LIN {X -0.043,Y -388.097,Z 1443.709,A 0.000,B 0.000,C 90.000,E1 163.614} C_DIS
LIN {X -0.106,Y -389.112,Z 1443.709,A 0.000,B 0.000,C 90.000,E1 163.614} C_DIS
LIN {X 0.170,Y -391.805,Z 1443.708,A 0.000,B 0.000,C 90.000,E1 163.504} C_DIS
LIN {X 0.071,Y -393.632,Z 1443.708,A 0.000,B 0.000,C 90.000,E1 163.449} C_DIS
LIN {X 0.005,Y -396.516,Z 1443.707,A 0.000,B 0.000,C 90.000,E1 163.323} C_DIS
LIN {X 0.115,Y -399.461,Z 1443.707,A 0.000,B 0.000,C 90.000,E1 163.142} C_DIS
LIN {X -0.176,Y -405.694,Z 1443.704,A 0.000,B 0.000,C 90.000,E1 162.779} C_DIS
LIN {X -0.149,Y -411.913,Z 1443.702,A 0.000,B 0.000,C 90.000,E1 162.308} C_DIS
LIN {X 0.069,Y -418.024,Z 1443.699,A 0.000,B 0.000,C 90.000,E1 161.764} C_DIS
LIN {X -0.143,Y -430.224,Z 1443.693,A 0.000,B 0.000,C 90.000,E1 160.732} C_DIS
LIN {X 0.007,Y -445.761,Z 1443.686,A 0.000,B 0.000,C 90.000,E1 159.390} C_DIS
LIN {X 0.043,Y -457.905,Z 1443.680,A 0.000,B 0.000,C 90.000,E1 158.358} C_DIS
LIN {X -0.134,Y -466.994,Z 1443.676,A 0.000,B 0.000,C 90.000,E1 157.614} C_DIS
LIN {X 0.217,Y -474.540,Z 1443.672,A 0.000,B 0.000,C 90.000,E1 156.922} C_DIS
LIN {X -0.067,Y -483.447,Z 1443.668,A 0.000,B 0.000,C 90.000,E1 156.177} C_DIS
LIN {X 0.031,Y -493.492,Z 1443.662,A 0.000,B 0.000,C 90.000,E1 155.229} C_DIS
LIN {X 0.119,Y -500.398,Z 1443.659,A 0.000,B 0.000,C 90.000,E1 154.537} C_DIS
LIN {X -0.168,Y -505.638,Z 1443.656,A 0.000,B 0.000,C 90.000,E1 154.024} C_DIS
LIN {X -0.036,Y -510.716,Z 1443.652,A 0.000,B 0.000,C 90.000,E1 153.435} C_DIS
LIN {X -0.076,Y -514.384,Z 1443.650,A 0.000,B 0.000,C 90.000,E1 152.999} C_DIS
LIN {X -0.071,Y -518.865,Z 1443.647,A 0.000,B 0.000,C 90.000,E1 152.410} C_DIS
LIN {X -0.031,Y -522.887,Z 1443.643,A 0.000,B 0.000,C 90.000,E1 151.820} C_DIS
LIN {X -0.114,Y -527.207,Z 1443.639,A 0.000,B 0.000,C 90.000,E1 151.101} C_DIS
LIN {X -0.010,Y -530.289,Z 1443.636,A 0.000,B 0.000,C 90.000,E1 150.511} C_DIS
LIN {X -0.030,Y -533.682,Z 1443.632,A 0.000,B 0.000,C 90.000,E1 149.793} C_DIS
LIN {X 0.121,Y -536.153,Z 1443.629,A 0.000,B 0.000,C 90.000,E1 149.203} C_DIS
LIN {X -0.174,Y -538.356,Z 1443.626,A 0.000,B 0.000,C 90.000,E1 148.663} C_DIS
LIN {X 0.009,Y -541.283,Z 1443.621,A 0.000,B 0.000,C 90.000,E1 147.788} C_DIS
LIN {X 0.224,Y -543.843,Z 1443.616,A 0.000,B 0.000,C 90.000,E1 146.914} C_DIS
LIN {X 0.045,Y -546.875,Z 1443.610,A 0.000,B 0.000,C 90.000,E1 145.801} C_DIS
LIN {X -0.138,Y -548.886,Z 1443.605,A 0.000,B 0.000,C 90.000,E1 144.975} C_DIS
LIN {X -0.039,Y -550.081,Z 1443.602,A 0.000,B 0.000,C 90.000,E1 144.402} C_DIS
LIN {X 0.133,Y -551.642,Z 1443.598,A 0.000,B 0.000,C 90.000,E1 143.543} C_DIS
LIN {X -0.012,Y -552.949,Z 1443.593,A 0.000,B 0.000,C 90.000,E1 142.718} C_DIS
LIN {X -0.183,Y -554.507,Z 1443.587,A 0.000,B 0.000,C 90.000,E1 141.618} C_DIS
LIN {X 0.027,Y -555.474,Z 1443.582,A 0.000,B 0.000,C 90.000,E1 140.759} C_DIS
LIN {X -0.106,Y -556.824,Z 1443.574,A 0.000,B 0.000,C 90.000,E1 139.380} C_DIS
LIN {X -0.132,Y -558.199,Z 1443.565,A 0.000,B 0.000,C 90.000,E1 137.715} C_DIS
LIN {X 0.168,Y -559.249,Z 1443.557,A 0.000,B 0.000,C 90.000,E1 136.296} C_DIS
LIN {X 0.023,Y -559.895,Z 1443.551,A 0.000,B 0.000,C 90.000,E1 135.202} C_DIS
LIN {X 0.216,Y -560.297,Z 1443.547,A 0.000,B 0.000,C 90.000,E1 134.352} C_DIS
LIN {X -0.236,Y -560.810,Z 1443.539,A 0.000,B 0.000,C 90.000,E1 133.014} C_DIS
LIN {X 0.023,Y -561.097,Z 1443.533,A 0.000,B 0.000,C 90.000,E1 131.881} C_DIS
LIN {X 0.076,Y -561.154,Z 1443.524,A 0.000,B 0.000,C 90.000,E1 130.216} C_DIS
LIN {X 0.112,Y -561.234,Z 1443.516,A 0.000,B 0.000,C 90.000,E1 128.830} C_DIS
LIN {X 0.155,Y -561.226,Z 1443.508,A 0.000,B 0.000,C 90.000,E1 127.443} C_DIS
LIN {X -0.142,Y -561.158,Z 1443.500,A 0.000,B 0.000,C 90.000,E1 126.091} C_DIS
LIN {X 0.113,Y -560.907,Z 1443.491,A 0.000,B 0.000,C 90.000,E1 124.405} C_DIS
LIN {X -0.047,Y -560.612,Z 1443.484,A 0.000,B 0.000,C 90.000,E1 123.038} C_DIS
LIN {X 0.013,Y -560.329,Z 1443.470,A 0.000,B 0.000,C 90.000,E1 120.541} C_DIS
LIN {X 0.051,Y -560.806,Z 1443.454,A 0.000,B 0.000,C 90.000,E1 117.769} C_DIS
LIN {X -0.092,Y -561.432,Z 1443.444,A 0.000,B 0.000,C 90.000,E1 115.848} C_DIS
LIN {X -0.264,Y -561.973,Z 1443.434,A 0.000,B 0.000,C 90.000,E1 114.207} C_DIS
LIN {X 0.286,Y -562.387,Z 1443.427,A 0.000,B 0.000,C 90.000,E1 112.770} C_DIS
LIN {X 0.020,Y -563.124,Z 1443.416,A 0.000,B 0.000,C 90.000,E1 110.865} C_DIS
LIN {X -0.155,Y -563.887,Z 1443.408,A 0.000,B 0.000,C 90.000,E1 109.504} C_DIS
LIN {X 0.195,Y -564.616,Z 1443.405,A 0.000,B 0.000,C 90.000,E1 108.779} C_DIS
LIN {X -0.178,Y -565.734,Z 1443.402,A 0.000,B 0.000,C 90.000,E1 108.362} C_DIS
LIN {X 0.147,Y -567.188,Z 1443.400,A 0.000,B 0.000,C 90.000,E1 108.055} C_DIS
LIN {X -0.135,Y -568.209,Z 1443.400,A 0.000,B 0.000,C 90.000,E1 107.946} C_DIS
LIN {X 0.222,Y -571.023,Z 1443.398,A 0.000,B 0.000,C 90.000,E1 107.638} C_DIS
LIN {X -0.047,Y -580.628,Z 1443.394,A 0.000,B 0.000,C 90.000,E1 106.913} C_DIS
LIN {X 0.055,Y -584.581,Z 1443.392,A 0.000,B 0.000,C 90.000,E1 106.551} C_DIS
LIN {X -0.083,Y -587.115,Z 1443.391,A 0.000,B 0.000,C 90.000,E1 106.315} C_DIS
LIN {X -0.078,Y -591.677,Z 1443.388,A 0.000,B 0.000,C 90.000,E1 105.788} C_DIS
LIN {X -0.155,Y -592.571,Z 1443.387,A 0.000,B 0.000,C 90.000,E1 105.662} C_DIS
LIN {X -0.267,Y -596.101,Z 1443.383,A 0.000,B 0.000,C 90.000,E1 105.009} C_DIS
LIN {X 0.237,Y -596.677,Z 1443.383,A 0.000,B 0.000,C 90.000,E1 104.828} C_DIS
LIN {X 0.228,Y -597.980,Z 1443.380,A 0.000,B 0.000,C 90.000,E1 104.300} C_DIS
LIN {X -0.055,Y -599.497,Z 1443.375,A 0.000,B 0.000,C 90.000,E1 103.536} C_DIS
LIN {X -0.039,Y -600.150,Z 1443.372,A 0.000,B 0.000,C 90.000,E1 103.008} C_DIS
LIN {X -0.297,Y -600.745,Z 1443.368,A 0.000,B 0.000,C 90.000,E1 102.243} C_DIS
LIN {X 0.035,Y -600.724,Z 1443.364,A 0.000,B 0.000,C 90.000,E1 101.422} C_DIS
LIN {X -0.247,Y -600.676,Z 1443.362,A 0.000,B 0.000,C 90.000,E1 101.186} C_DIS
LIN {X -0.225,Y -599.926,Z 1443.359,A 0.000,B 0.000,C 90.000,E1 100.658} C_DIS
LIN {X -0.315,Y -598.816,Z 1443.356,A 0.000,B 0.000,C 90.000,E1 100.141} C_DIS
LIN {X -0.013,Y -598.181,Z 1443.355,A 0.000,B 0.000,C 90.000,E1 99.849} C_DIS
LIN {X -0.011,Y -596.569,Z 1443.352,A 0.000,B 0.000,C 90.000,E1 99.321} C_DIS
LIN {X -0.223,Y -593.855,Z 1443.348,A 0.000,B 0.000,C 90.000,E1 98.681} C_DIS
LIN {X 0.239,Y -591.207,Z 1443.345,A 0.000,B 0.000,C 90.000,E1 98.106} C_DIS
LIN {X 0.100,Y -588.095,Z 1443.342,A 0.000,B 0.000,C 90.000,E1 97.587} C_DIS
LIN {X -0.191,Y -583.595,Z 1443.339,A 0.000,B 0.000,C 90.000,E1 96.947} C_DIS
LIN {X 0.198,Y -579.504,Z 1443.336,A 0.000,B 0.000,C 90.000,E1 96.372} C_DIS
LIN {X -0.018,Y -574.862,Z 1443.333,A 0.000,B 0.000,C 90.000,E1 95.853} C_DIS
LIN {X -0.099,Y -572.597,Z 1443.330,A 0.000,B 0.000,C 90.000,E1 95.454} C_DIS
LIN {X 0.195,Y -571.361,Z 1443.329,A 0.000,B 0.000,C 90.000,E1 95.220} C_DIS
LIN {X 0.085,Y -571.073,Z 1443.329,A 0.000,B 0.000,C 90.000,E1 95.163} C_DIS
LIN {X 0.211,Y -570.540,Z 1443.327,A 0.000,B 0.000,C 90.000,E1 94.878} C_DIS
LIN {X -0.137,Y -570.023,Z 1443.324,A 0.000,B 0.000,C 90.000,E1 94.302} C_DIS
LIN {X 0.276,Y -570.225,Z 1443.319,A 0.000,B 0.000,C 90.000,E1 93.440} C_DIS
LIN {X -0.056,Y -571.455,Z 1443.310,A 0.000,B 0.000,C 90.000,E1 91.835} C_DIS
LIN {X -0.225,Y -573.087,Z 1443.300,A 0.000,B 0.000,C 90.000,E1 89.943} C_DIS
LIN {X -0.209,Y -575.053,Z 1443.287,A 0.000,B 0.000,C 90.000,E1 87.764} C_DIS
LIN {X -0.114,Y -577.038,Z 1443.276,A 0.000,B 0.000,C 90.000,E1 85.584} C_DIS
LIN {X 0.129,Y -579.039,Z 1443.263,A 0.000,B 0.000,C 90.000,E1 83.394} C_DIS
LIN {X -0.084,Y -580.371,Z 1443.256,A 0.000,B 0.000,C 90.000,E1 82.064} C_DIS
LIN {X -0.280,Y -581.712,Z 1443.248,A 0.000,B 0.000,C 90.000,E1 80.735} C_DIS
LIN {X -0.228,Y -583.857,Z 1443.236,A 0.000,B 0.000,C 90.000,E1 78.578} C_DIS
LIN {X 0.166,Y -584.968,Z 1443.230,A 0.000,B 0.000,C 90.000,E1 77.465} C_DIS
LIN {X 0.165,Y -586.431,Z 1443.220,A 0.000,B 0.000,C 90.000,E1 75.589} C_DIS
LIN {X 0.159,Y -587.187,Z 1443.214,A 0.000,B 0.000,C 90.000,E1 74.519} C_DIS
LIN {X 0.251,Y -588.124,Z 1443.205,A 0.000,B 0.000,C 90.000,E1 72.906} C_DIS
LIN {X -0.116,Y -588.784,Z 1443.199,A 0.000,B 0.000,C 90.000,E1 71.873} C_DIS
LIN {X -0.133,Y -589.718,Z 1443.189,A 0.000,B 0.000,C 90.000,E1 70.007} C_DIS
LIN {X 0.155,Y -590.890,Z 1443.177,A 0.000,B 0.000,C 90.000,E1 67.847} C_DIS
LIN {X -0.064,Y -591.621,Z 1443.170,A 0.000,B 0.000,C 90.000,E1 66.538} C_DIS
LIN {X -0.321,Y -593.633,Z 1443.153,A 0.000,B 0.000,C 90.000,E1 63.640} C_DIS
LIN {X -0.075,Y -594.193,Z 1443.149,A 0.000,B 0.000,C 90.000,E1 62.820} C_DIS
LIN {X -0.243,Y -595.838,Z 1443.137,A 0.000,B 0.000,C 90.000,E1 60.717} C_DIS
LIN {X -0.306,Y -596.762,Z 1443.131,A 0.000,B 0.000,C 90.000,E1 59.665} C_DIS
LIN {X -0.143,Y -597.955,Z 1443.124,A 0.000,B 0.000,C 90.000,E1 58.329} C_DIS
LIN {X 0.128,Y -598.911,Z 1443.118,A 0.000,B 0.000,C 90.000,E1 57.248} C_DIS
LIN {X 0.052,Y -600.312,Z 1443.109,A 0.000,B 0.000,C 90.000,E1 55.674} C_DIS
LIN {X -0.149,Y -601.697,Z 1443.101,A 0.000,B 0.000,C 90.000,E1 54.116} C_DIS
LIN {X -0.067,Y -602.999,Z 1443.090,A 0.000,B 0.000,C 90.000,E1 52.271} C_DIS
LIN {X -0.370,Y -603.736,Z 1443.085,A 0.000,B 0.000,C 90.000,E1 51.251} C_DIS
LIN {X 0.233,Y -604.562,Z 1443.076,A 0.000,B 0.000,C 90.000,E1 49.622} C_DIS
LIN {X -0.121,Y -604.812,Z 1443.070,A 0.000,B 0.000,C 90.000,E1 48.609} C_DIS
LIN {X -0.165,Y -605.143,Z 1443.060,A 0.000,B 0.000,C 90.000,E1 46.782} C_DIS
LIN {X -0.285,Y -605.195,Z 1443.053,A 0.000,B 0.000,C 90.000,E1 45.486} C_DIS
LIN {X 0.183,Y -605.142,Z 1443.050,A 0.000,B 0.000,C 90.000,E1 44.919} C_DIS
LIN {X -0.399,Y -604.870,Z 1443.045,A 0.000,B 0.000,C 90.000,E1 44.190} C_DIS
LIN {X 0.112,Y -604.301,Z 1443.040,A 0.000,B 0.000,C 90.000,E1 43.095} C_DIS
LIN {X 0.413,Y -603.357,Z 1443.032,A 0.000,B 0.000,C 90.000,E1 41.757} C_DIS
LIN {X 0.249,Y -602.682,Z 1443.028,A 0.000,B 0.000,C 90.000,E1 40.987} C_DIS
LIN {X -0.065,Y -601.561,Z 1443.022,A 0.000,B 0.000,C 90.000,E1 39.967} C_DIS
LIN {X -0.227,Y -599.921,Z 1443.015,A 0.000,B 0.000,C 90.000,E1 38.669} C_DIS
LIN {X -0.098,Y -598.436,Z 1443.009,A 0.000,B 0.000,C 90.000,E1 37.604} C_DIS
LIN {X 0.139,Y -597.159,Z 1443.005,A 0.000,B 0.000,C 90.000,E1 36.790} C_DIS
LIN {X 0.231,Y -595.164,Z 1442.999,A 0.000,B 0.000,C 90.000,E1 35.724} C_DIS
LIN {X 0.073,Y -593.383,Z 1442.994,A 0.000,B 0.000,C 90.000,E1 34.945} C_DIS
LIN {X -0.230,Y -590.841,Z 1442.988,A 0.000,B 0.000,C 90.000,E1 33.913} C_DIS
LIN {X -0.069,Y -587.912,Z 1442.982,A 0.000,B 0.000,C 90.000,E1 32.832} C_DIS
LIN {X 0.183,Y -585.485,Z 1442.978,A 0.000,B 0.000,C 90.000,E1 32.005} C_DIS
LIN {X 0.232,Y -583.740,Z 1442.975,A 0.000,B 0.000,C 90.000,E1 31.465} C_DIS
LIN {X 0.130,Y -580.685,Z 1442.970,A 0.000,B 0.000,C 90.000,E1 30.669} C_DIS
LIN {X 0.072,Y -577.807,Z 1442.967,A 0.000,B 0.000,C 90.000,E1 30.001} C_DIS
LIN {X -0.173,Y -573.342,Z 1442.962,A 0.000,B 0.000,C 90.000,E1 29.077} C_DIS
LIN {X 0.197,Y -569.830,Z 1442.958,A 0.000,B 0.000,C 90.000,E1 28.359} C_DIS
LIN {X -0.146,Y -566.821,Z 1442.955,A 0.000,B 0.000,C 90.000,E1 27.847} C_DIS
LIN {X -0.028,Y -561.226,Z 1442.949,A 0.000,B 0.000,C 90.000,E1 26.873} C_DIS
LIN {X -0.127,Y -556.006,Z 1442.945,A 0.000,B 0.000,C 90.000,E1 26.052} C_DIS
LIN {X 0.293,Y -553.280,Z 1442.942,A 0.000,B 0.000,C 90.000,E1 25.591} C_DIS
LIN {X -0.156,Y -549.389,Z 1442.939,A 0.000,B 0.000,C 90.000,E1 25.079} C_DIS
LIN {X 0.242,Y -544.155,Z 1442.935,A 0.000,B 0.000,C 90.000,E1 24.335} C_DIS
LIN {X -0.138,Y -540.821,Z 1442.933,A 0.000,B 0.000,C 90.000,E1 23.951} C_DIS
LIN {X 0.182,Y -534.920,Z 1442.929,A 0.000,B 0.000,C 90.000,E1 23.206} C_DIS
LIN {X -0.196,Y -527.495,Z 1442.924,A 0.000,B 0.000,C 90.000,E1 22.386} C_DIS
LIN {X 0.203,Y -518.579,Z 1442.919,A 0.000,B 0.000,C 90.000,E1 21.354} C_DIS
LIN {X 0.160,Y -509.329,Z 1442.913,A 0.000,B 0.000,C 90.000,E1 20.375} C_DIS
LIN {X -0.060,Y -498.393,Z 1442.907,A 0.000,B 0.000,C 90.000,E1 19.268} C_DIS
LIN {X 0.009,Y -478.216,Z 1442.895,A 0.000,B 0.000,C 90.000,E1 17.166} C_DIS
LIN {X 0.259,Y -464.739,Z 1442.887,A 0.000,B 0.000,C 90.000,E1 15.662} C_DIS
LIN {X 0.014,Y -460.341,Z 1442.885,A 0.000,B 0.000,C 90.000,E1 15.245} C_DIS
LIN {X -0.012,Y -455.773,Z 1442.882,A 0.000,B 0.000,C 90.000,E1 14.828} C_DIS
LIN {X 0.032,Y -450.844,Z 1442.880,A 0.000,B 0.000,C 90.000,E1 14.426} C_DIS
LIN {X 0.002,Y -447.084,Z 1442.879,A 0.000,B 0.000,C 90.000,E1 14.189} C_DIS
LIN {X 0.033,Y -444.395,Z 1442.878,A 0.000,B 0.000,C 90.000,E1 14.064} C_DIS
LIN {X 0.098,Y -442.520,Z 1442.878,A 0.000,B 0.000,C 90.000,E1 14.008} C_DIS
LIN {X 0.070,Y -442.170,Z 1442.878,A 0.000,B 0.000,C 90.000,E1 14.008} C_DIS
LIN {X 0.034,Y -369.502,Z 1442.878,A 0.000,B 0.000,C 90.000,E1 14.008} C_DIS
LIN {X 0.102,Y -366.485,Z 1442.855,A 0.000,B 0.000,C 90.000,E1 9.905} C_DIS
LIN {X 0.038,Y -361.787,Z 1442.822,A 0.000,B 0.000,C 90.000,E1 3.955} C_DIS
LIN {X -0.077,Y -360.901,Z 1442.801,A 0.000,B 0.000,C 90.000,E1 0.229} C_DIS
LIN {X -0.053,Y -359.426,Z 1442.770,A 0.000,B 0.000,C 90.000,E1 354.546} C_DIS
LIN {X 0.070,Y -358.890,Z 1442.759,A 0.000,B 0.000,C 90.000,E1 352.648} C_DIS
LIN {X -0.020,Y -359.563,Z 1442.726,A 0.000,B 0.000,C 90.000,E1 346.645} C_DIS
LIN {X 0.001,Y -361.801,Z 1442.684,A 0.000,B 0.000,C 90.000,E1 339.135} C_DIS
LIN {X -0.154,Y -362.053,Z 1442.680,A 0.000,B 0.000,C 90.000,E1 338.411} C_DIS
LIN {X 0.189,Y -365.980,Z 1442.643,A 0.000,B 0.000,C 90.000,E1 331.641} C_DIS
LIN {X 0.029,Y -366.387,Z 1442.639,A 0.000,B 0.000,C 90.000,E1 330.923} C_DIS
LIN {X -0.031,Y -371.355,Z 1442.604,A 0.000,B 0.000,C 90.000,E1 324.642} C_DIS
LIN {X -0.043,Y -371.766,Z 1442.602,A 0.000,B 0.000,C 90.000,E1 324.276} C_DIS
LIN {X 0.013,Y -377.358,Z 1442.567,A 0.000,B 0.000,C 90.000,E1 318.038} C_DIS
LIN {X 0.012,Y -378.235,Z 1442.563,A 0.000,B 0.000,C 90.000,E1 317.310} C_DIS
LIN {X 0.002,Y -383.940,Z 1442.531,A 0.000,B 0.000,C 90.000,E1 311.515} C_DIS
LIN {X 0.088,Y -384.893,Z 1442.527,A 0.000,B 0.000,C 90.000,E1 310.782} C_DIS
LIN {X 0.262,Y -390.610,Z 1442.495,A 0.000,B 0.000,C 90.000,E1 305.025} C_DIS
LIN {X 0.106,Y -391.104,Z 1442.493,A 0.000,B 0.000,C 90.000,E1 304.692} C_DIS
LIN {X 0.022,Y -391.648,Z 1442.489,A 0.000,B 0.000,C 90.000,E1 303.992} C_DIS
LIN {X -0.080,Y -396.825,Z 1442.459,A 0.000,B 0.000,C 90.000,E1 298.693} C_DIS
LIN {X -0.210,Y -397.120,Z 1442.457,A 0.000,B 0.000,C 90.000,E1 298.359} C_DIS
LIN {X -0.055,Y -401.597,Z 1442.426,A 0.000,B 0.000,C 90.000,E1 292.717} C_DIS
LIN {X 0.222,Y -404.659,Z 1442.395,A 0.000,B 0.000,C 90.000,E1 287.094} C_DIS
LIN {X -0.079,Y -404.735,Z 1442.391,A 0.000,B 0.000,C 90.000,E1 286.441} C_DIS
LIN {X 0.214,Y -406.099,Z 1442.364,A 0.000,B 0.000,C 90.000,E1 281.535} C_DIS
LIN {X -0.176,Y -406.094,Z 1442.362,A 0.000,B 0.000,C 90.000,E1 281.243} C_DIS
LIN {X -0.097,Y -405.680,Z 1442.333,A 0.000,B 0.000,C 90.000,E1 276.024} C_DIS
LIN {X -0.165,Y -405.058,Z 1442.328,A 0.000,B 0.000,C 90.000,E1 274.992} C_DIS
LIN {X -0.060,Y -403.497,Z 1442.304,A 0.000,B 0.000,C 90.000,E1 270.802} C_DIS
LIN {X -0.092,Y -403.288,Z 1442.302,A 0.000,B 0.000,C 90.000,E1 270.458} C_DIS
LIN {X 0.091,Y -398.931,Z 1442.271,A 0.000,B 0.000,C 90.000,E1 264.837} C_DIS
LIN {X -0.040,Y -393.108,Z 1442.242,A 0.000,B 0.000,C 90.000,E1 259.567} C_DIS
LIN {X -0.079,Y -392.835,Z 1442.240,A 0.000,B 0.000,C 90.000,E1 259.218} C_DIS
LIN {X 0.034,Y -385.993,Z 1442.212,A 0.000,B 0.000,C 90.000,E1 254.212} C_DIS
LIN {X -0.026,Y -385.267,Z 1442.208,A 0.000,B 0.000,C 90.000,E1 253.504} C_DIS
LIN {X -0.004,Y -384.768,Z 1442.206,A 0.000,B 0.000,C 90.000,E1 253.142} C_DIS
LIN {X 0.221,Y -377.973,Z 1442.182,A 0.000,B 0.000,C 90.000,E1 248.773} C_DIS
LIN {X -0.044,Y -376.233,Z 1442.174,A 0.000,B 0.000,C 90.000,E1 247.358} C_DIS
LIN {X 0.057,Y -374.944,Z 1442.170,A 0.000,B 0.000,C 90.000,E1 246.613} C_DIS
LIN {X -0.208,Y -368.417,Z 1442.148,A 0.000,B 0.000,C 90.000,E1 242.615} C_DIS
LIN {X 0.097,Y -366.047,Z 1442.137,A 0.000,B 0.000,C 90.000,E1 240.717} C_DIS
LIN {X 0.004,Y -359.196,Z 1442.115,A 0.000,B 0.000,C 90.000,E1 236.628} C_DIS
LIN {X 0.021,Y -355.842,Z 1442.100,A 0.000,B 0.000,C 90.000,E1 233.989} C_DIS
LIN {X -0.173,Y -348.793,Z 1442.075,A 0.000,B 0.000,C 90.000,E1 229.461} C_DIS
LIN {X -0.097,Y -346.185,Z 1442.062,A 0.000,B 0.000,C 90.000,E1 227.148} C_DIS
LIN {X -0.088,Y -345.065,Z 1442.058,A 0.000,B 0.000,C 90.000,E1 226.377} C_DIS
LIN {X 0.094,Y -338.586,Z 1442.030,A 0.000,B 0.000,C 90.000,E1 221.310} C_DIS
LIN {X 0.094,Y -336.840,Z 1442.019,A 0.000,B 0.000,C 90.000,E1 219.358} C_DIS
LIN {X 0.014,Y -330.861,Z 1441.988,A 0.000,B 0.000,C 90.000,E1 213.865} C_DIS
LIN {X 0.149,Y -329.296,Z 1441.975,A 0.000,B 0.000,C 90.000,E1 211.465} C_DIS
LIN {X -0.154,Y -324.669,Z 1441.942,A 0.000,B 0.000,C 90.000,E1 205.540} C_DIS
LIN {X 0.174,Y -323.837,Z 1441.928,A 0.000,B 0.000,C 90.000,E1 203.078} C_DIS
LIN {X -0.017,Y -321.124,Z 1441.881,A 0.000,B 0.000,C 90.000,E1 194.662} C_DIS
LIN {X 0.138,Y -320.932,Z 1441.877,A 0.000,B 0.000,C 90.000,E1 193.828} C_DIS
LIN {X -0.076,Y -321.562,Z 1441.832,A 0.000,B 0.000,C 90.000,E1 185.796} C_DIS
LIN {X -0.143,Y -324.415,Z 1441.790,A 0.000,B 0.000,C 90.000,E1 178.165} C_DIS
LIN {X -0.141,Y -325.376,Z 1441.783,A 0.000,B 0.000,C 90.000,E1 176.963} C_DIS
LIN {X -0.100,Y -329.112,Z 1441.750,A 0.000,B 0.000,C 90.000,E1 170.971} C_DIS
LIN {X 0.061,Y -334.260,Z 1441.726,A 0.000,B 0.000,C 90.000,E1 166.589} C_DIS
LIN {X 0.067,Y -335.488,Z 1441.719,A 0.000,B 0.000,C 90.000,E1 165.408} C_DIS
LIN {X -0.119,Y -336.681,Z 1441.713,A 0.000,B 0.000,C 90.000,E1 164.338} C_DIS
LIN {X -0.154,Y -381.447,Z 1441.713,A 0.000,B 0.000,C 90.000,E1 164.338} C_DIS
LIN {X 0.204,Y -384.725,Z 1441.713,A 0.000,B 0.000,C 90.000,E1 164.212} C_DIS
LIN {X -0.022,Y -386.911,Z 1441.712,A 0.000,B 0.000,C 90.000,E1 164.157} C_DIS
LIN {X -0.146,Y -389.736,Z 1441.711,A 0.000,B 0.000,C 90.000,E1 164.031} C_DIS
LIN {X 0.097,Y -395.861,Z 1441.709,A 0.000,B 0.000,C 90.000,E1 163.614} C_DIS
LIN {X -0.141,Y -402.081,Z 1441.707,A 0.000,B 0.000,C 90.000,E1 163.196} C_DIS
LIN {X 0.031,Y -408.356,Z 1441.704,A 0.000,B 0.000,C 90.000,E1 162.670} C_DIS
LIN {X 0.045,Y -422.169,Z 1441.697,A 0.000,B 0.000,C 90.000,E1 161.456} C_DIS
LIN {X -0.198,Y -434.491,Z 1441.691,A 0.000,B 0.000,C 90.000,E1 160.423} C_DIS
LIN {X 0.067,Y -448.418,Z 1441.685,A 0.000,B 0.000,C 90.000,E1 159.209} C_DIS
LIN {X 0.281,Y -460.594,Z 1441.679,A 0.000,B 0.000,C 90.000,E1 158.156} C_DIS
LIN {X -0.085,Y -471.156,Z 1441.674,A 0.000,B 0.000,C 90.000,E1 157.305} C_DIS
LIN {X 0.223,Y -483.026,Z 1441.668,A 0.000,B 0.000,C 90.000,E1 156.230} C_DIS
LIN {X -0.253,Y -491.639,Z 1441.664,A 0.000,B 0.000,C 90.000,E1 155.485} C_DIS
LIN {X -0.063,Y -497.243,Z 1441.661,A 0.000,B 0.000,C 90.000,E1 154.921} C_DIS
LIN {X 0.015,Y -502.740,Z 1441.658,A 0.000,B 0.000,C 90.000,E1 154.357} C_DIS
LIN {X -0.077,Y -506.692,Z 1441.655,A 0.000,B 0.000,C 90.000,E1 153.948} C_DIS
LIN {X -0.161,Y -511.719,Z 1441.652,A 0.000,B 0.000,C 90.000,E1 153.384} C_DIS
LIN {X -0.003,Y -515.332,Z 1441.650,A 0.000,B 0.000,C 90.000,E1 152.922} C_DIS
LIN {X -0.229,Y -519.733,Z 1441.646,A 0.000,B 0.000,C 90.000,E1 152.359} C_DIS
LIN {X -0.186,Y -523.691,Z 1441.643,A 0.000,B 0.000,C 90.000,E1 151.769} C_DIS
LIN {X -0.110,Y -527.162,Z 1441.640,A 0.000,B 0.000,C 90.000,E1 151.179} C_DIS
LIN {X -0.008,Y -530.281,Z 1441.637,A 0.000,B 0.000,C 90.000,E1 150.589} C_DIS
LIN {X -0.030,Y -533.716,Z 1441.633,A 0.000,B 0.000,C 90.000,E1 149.871} C_DIS
LIN {X 0.118,Y -536.208,Z 1441.630,A 0.000,B 0.000,C 90.000,E1 149.282} C_DIS
LIN {X -0.179,Y -538.438,Z 1441.626,A 0.000,B 0.000,C 90.000,E1 148.742} C_DIS
LIN {X 0.003,Y -541.355,Z 1441.622,A 0.000,B 0.000,C 90.000,E1 147.867} C_DIS
LIN {X -0.240,Y -543.932,Z 1441.617,A 0.000,B 0.000,C 90.000,E1 147.041} C_DIS
LIN {X 0.036,Y -546.954,Z 1441.610,A 0.000,B 0.000,C 90.000,E1 145.881} C_DIS
LIN {X -0.149,Y -548.980,Z 1441.606,A 0.000,B 0.000,C 90.000,E1 145.055} C_DIS
LIN {X 0.003,Y -550.716,Z 1441.601,A 0.000,B 0.000,C 90.000,E1 144.196} C_DIS
LIN {X 0.181,Y -552.207,Z 1441.596,A 0.000,B 0.000,C 90.000,E1 143.336} C_DIS
LIN {X -0.333,Y -553.829,Z 1441.590,A 0.000,B 0.000,C 90.000,E1 142.271} C_DIS
LIN {X 0.292,Y -555.266,Z 1441.584,A 0.000,B 0.000,C 90.000,E1 141.090} C_DIS
LIN {X -0.195,Y -556.619,Z 1441.576,A 0.000,B 0.000,C 90.000,E1 139.747} C_DIS
LIN {X -0.220,Y -558.014,Z 1441.567,A 0.000,B 0.000,C 90.000,E1 138.081} C_DIS
LIN {X 0.081,Y -559.071,Z 1441.559,A 0.000,B 0.000,C 90.000,E1 136.662} C_DIS
LIN {X -0.058,Y -559.788,Z 1441.553,A 0.000,B 0.000,C 90.000,E1 135.567} C_DIS
LIN {X 0.201,Y -560.311,Z 1441.547,A 0.000,B 0.000,C 90.000,E1 134.433} C_DIS
LIN {X 0.132,Y -560.797,Z 1441.539,A 0.000,B 0.000,C 90.000,E1 133.056} C_DIS
LIN {X -0.035,Y -561.010,Z 1441.535,A 0.000,B 0.000,C 90.000,E1 132.243} C_DIS
LIN {X -0.149,Y -561.120,Z 1441.529,A 0.000,B 0.000,C 90.000,E1 131.148} C_DIS
LIN {X 0.005,Y -561.229,Z 1441.518,A 0.000,B 0.000,C 90.000,E1 129.197} C_DIS
LIN {X 0.049,Y -561.246,Z 1441.510,A 0.000,B 0.000,C 90.000,E1 127.810} C_DIS
LIN {X -0.148,Y -561.170,Z 1441.501,A 0.000,B 0.000,C 90.000,E1 126.171} C_DIS
LIN {X 0.204,Y -560.871,Z 1441.490,A 0.000,B 0.000,C 90.000,E1 124.199} C_DIS
LIN {X 0.045,Y -560.558,Z 1441.482,A 0.000,B 0.000,C 90.000,E1 122.832} C_DIS
LIN {X -0.106,Y -560.332,Z 1441.467,A 0.000,B 0.000,C 90.000,E1 120.079} C_DIS
LIN {X -0.129,Y -560.864,Z 1441.453,A 0.000,B 0.000,C 90.000,E1 117.590} C_DIS
LIN {X -0.019,Y -561.513,Z 1441.443,A 0.000,B 0.000,C 90.000,E1 115.643} C_DIS
LIN {X 0.001,Y -561.999,Z 1441.435,A 0.000,B 0.000,C 90.000,E1 114.259} C_DIS
LIN {X -0.190,Y -562.387,Z 1441.427,A 0.000,B 0.000,C 90.000,E1 112.898} C_DIS
LIN {X 0.068,Y -563.266,Z 1441.415,A 0.000,B 0.000,C 90.000,E1 110.663} C_DIS
LIN {X -0.198,Y -564.236,Z 1441.408,A 0.000,B 0.000,C 90.000,E1 109.450} C_DIS
LIN {X 0.230,Y -564.662,Z 1441.407,A 0.000,B 0.000,C 90.000,E1 109.268} C_DIS
LIN {X 0.303,Y -565.625,Z 1441.405,A 0.000,B 0.000,C 90.000,E1 108.779} C_DIS
LIN {X 0.160,Y -566.006,Z 1441.404,A 0.000,B 0.000,C 90.000,E1 108.725} C_DIS
LIN {X -0.050,Y -568.089,Z 1441.403,A 0.000,B 0.000,C 90.000,E1 108.471} C_DIS
LIN {X 0.188,Y -572.870,Z 1441.401,A 0.000,B 0.000,C 90.000,E1 108.055} C_DIS
LIN {X -0.120,Y -577.443,Z 1441.399,A 0.000,B 0.000,C 90.000,E1 107.764} C_DIS
LIN {X -0.145,Y -582.962,Z 1441.396,A 0.000,B 0.000,C 90.000,E1 107.330} C_DIS
LIN {X -0.165,Y -588.165,Z 1441.394,A 0.000,B 0.000,C 90.000,E1 106.858} C_DIS
LIN {X 0.147,Y -592.829,Z 1441.391,A 0.000,B 0.000,C 90.000,E1 106.315} C_DIS
LIN {X -0.085,Y -593.845,Z 1441.390,A 0.000,B 0.000,C 90.000,E1 106.205} C_DIS
LIN {X -0.178,Y -598.056,Z 1441.386,A 0.000,B 0.000,C 90.000,E1 105.552} C_DIS
LIN {X -0.022,Y -600.169,Z 1441.383,A 0.000,B 0.000,C 90.000,E1 105.009} C_DIS
LIN {X 0.273,Y -601.137,Z 1441.382,A 0.000,B 0.000,C 90.000,E1 104.717} C_DIS
LIN {X -0.286,Y -602.332,Z 1441.379,A 0.000,B 0.000,C 90.000,E1 104.245} C_DIS
LIN {X 0.202,Y -603.643,Z 1441.375,A 0.000,B 0.000,C 90.000,E1 103.411} C_DIS
LIN {X 0.244,Y -604.336,Z 1441.372,A 0.000,B 0.000,C 90.000,E1 102.883} C_DIS
LIN {X 0.022,Y -604.816,Z 1441.367,A 0.000,B 0.000,C 90.000,E1 102.119} C_DIS
LIN {X 0.072,Y -604.770,Z 1441.365,A 0.000,B 0.000,C 90.000,E1 101.591} C_DIS
LIN {X 0.006,Y -604.432,Z 1441.362,A 0.000,B 0.000,C 90.000,E1 101.074} C_DIS
LIN {X 0.056,Y -603.692,Z 1441.359,A 0.000,B 0.000,C 90.000,E1 100.546} C_DIS
LIN {X 0.098,Y -602.585,Z 1441.356,A 0.000,B 0.000,C 90.000,E1 100.018} C_DIS
LIN {X -0.182,Y -601.937,Z 1441.354,A 0.000,B 0.000,C 90.000,E1 99.782} C_DIS
LIN {X -0.254,Y -600.334,Z 1441.351,A 0.000,B 0.000,C 90.000,E1 99.265} C_DIS
LIN {X -0.332,Y -598.273,Z 1441.349,A 0.000,B 0.000,C 90.000,E1 98.746} C_DIS
LIN {X 0.063,Y -595.130,Z 1441.345,A 0.000,B 0.000,C 90.000,E1 98.049} C_DIS
LIN {X -0.168,Y -591.288,Z 1441.341,A 0.000,B 0.000,C 90.000,E1 97.409} C_DIS
LIN {X 0.077,Y -587.188,Z 1441.337,A 0.000,B 0.000,C 90.000,E1 96.720} C_DIS
LIN {X 0.118,Y -584.208,Z 1441.335,A 0.000,B 0.000,C 90.000,E1 96.315} C_DIS
LIN {X -0.032,Y -578.292,Z 1441.332,A 0.000,B 0.000,C 90.000,E1 95.682} C_DIS
LIN {X 0.019,Y -574.437,Z 1441.329,A 0.000,B 0.000,C 90.000,E1 95.277} C_DIS
LIN {X -0.152,Y -573.540,Z 1441.329,A 0.000,B 0.000,C 90.000,E1 95.163} C_DIS
LIN {X 0.259,Y -571.279,Z 1441.326,A 0.000,B 0.000,C 90.000,E1 94.702} C_DIS
LIN {X 0.114,Y -570.398,Z 1441.323,A 0.000,B 0.000,C 90.000,E1 94.188} C_DIS
LIN {X -0.163,Y -570.247,Z 1441.320,A 0.000,B 0.000,C 90.000,E1 93.669} C_DIS
LIN {X -0.191,Y -570.844,Z 1441.314,A 0.000,B 0.000,C 90.000,E1 92.579} C_DIS
LIN {X 0.224,Y -571.549,Z 1441.310,A 0.000,B 0.000,C 90.000,E1 91.718} C_DIS
LIN {X 0.181,Y -573.409,Z 1441.298,A 0.000,B 0.000,C 90.000,E1 89.542} C_DIS
LIN {X 0.058,Y -575.156,Z 1441.287,A 0.000,B 0.000,C 90.000,E1 87.650} C_DIS
LIN {X 0.154,Y -577.155,Z 1441.275,A 0.000,B 0.000,C 90.000,E1 85.469} C_DIS
LIN {X -0.162,Y -578.372,Z 1441.267,A 0.000,B 0.000,C 90.000,E1 84.147} C_DIS
LIN {X -0.177,Y -580.001,Z 1441.258,A 0.000,B 0.000,C 90.000,E1 82.527} C_DIS
LIN {X -0.148,Y -581.636,Z 1441.249,A 0.000,B 0.000,C 90.000,E1 80.905} C_DIS
LIN {X -0.200,Y -583.766,Z 1441.237,A 0.000,B 0.000,C 90.000,E1 78.757} C_DIS
LIN {X -0.140,Y -585.134,Z 1441.230,A 0.000,B 0.000,C 90.000,E1 77.409} C_DIS
LIN {X 0.004,Y -586.584,Z 1441.220,A 0.000,B 0.000,C 90.000,E1 75.519} C_DIS
LIN {X 0.007,Y -587.341,Z 1441.214,A 0.000,B 0.000,C 90.000,E1 74.448} C_DIS
LIN {X -0.059,Y -588.287,Z 1441.205,A 0.000,B 0.000,C 90.000,E1 72.851} C_DIS
LIN {X 0.131,Y -588.918,Z 1441.199,A 0.000,B 0.000,C 90.000,E1 71.764} C_DIS
LIN {X 0.307,Y -589.855,Z 1441.188,A 0.000,B 0.000,C 90.000,E1 69.880} C_DIS
LIN {X -0.165,Y -591.048,Z 1441.177,A 0.000,B 0.000,C 90.000,E1 67.794} C_DIS
LIN {X 0.155,Y -591.771,Z 1441.169,A 0.000,B 0.000,C 90.000,E1 66.433} C_DIS
LIN {X -0.200,Y -593.344,Z 1441.156,A 0.000,B 0.000,C 90.000,E1 64.076} C_DIS
LIN {X 0.049,Y -594.058,Z 1441.151,A 0.000,B 0.000,C 90.000,E1 63.256} C_DIS
LIN {X 0.229,Y -596.043,Z 1441.137,A 0.000,B 0.000,C 90.000,E1 60.589} C_DIS
LIN {X 0.168,Y -596.956,Z 1441.131,A 0.000,B 0.000,C 90.000,E1 59.537} C_DIS
LIN {X -0.175,Y -598.169,Z 1441.124,A 0.000,B 0.000,C 90.000,E1 58.250} C_DIS
LIN {X 0.103,Y -599.105,Z 1441.118,A 0.000,B 0.000,C 90.000,E1 57.168} C_DIS
LIN {X -0.206,Y -600.297,Z 1441.110,A 0.000,B 0.000,C 90.000,E1 55.881} C_DIS
LIN {X 0.081,Y -601.656,Z 1441.102,A 0.000,B 0.000,C 90.000,E1 54.276} C_DIS
LIN {X 0.012,Y -602.633,Z 1441.094,A 0.000,B 0.000,C 90.000,E1 52.970} C_DIS
LIN {X -0.030,Y -603.591,Z 1441.087,A 0.000,B 0.000,C 90.000,E1 51.662} C_DIS
LIN {X 0.147,Y -604.200,Z 1441.081,A 0.000,B 0.000,C 90.000,E1 50.598} C_DIS
LIN {X 0.243,Y -604.751,Z 1441.075,A 0.000,B 0.000,C 90.000,E1 49.542} C_DIS
LIN {X 0.146,Y -605.014,Z 1441.068,A 0.000,B 0.000,C 90.000,E1 48.243} C_DIS
LIN {X -0.146,Y -605.295,Z 1441.059,A 0.000,B 0.000,C 90.000,E1 46.701} C_DIS
LIN {X -0.027,Y -605.352,Z 1441.051,A 0.000,B 0.000,C 90.000,E1 45.121} C_DIS
LIN {X -0.374,Y -604.988,Z 1441.045,A 0.000,B 0.000,C 90.000,E1 44.109} C_DIS
LIN {X 0.138,Y -604.421,Z 1441.039,A 0.000,B 0.000,C 90.000,E1 43.014} C_DIS
LIN {X 0.038,Y -603.496,Z 1441.032,A 0.000,B 0.000,C 90.000,E1 41.714} C_DIS
LIN {X -0.325,Y -602.554,Z 1441.026,A 0.000,B 0.000,C 90.000,E1 40.701} C_DIS
LIN {X -0.250,Y -601.351,Z 1441.020,A 0.000,B 0.000,C 90.000,E1 39.644} C_DIS
LIN {X 0.044,Y -599.704,Z 1441.013,A 0.000,B 0.000,C 90.000,E1 38.302} C_DIS
LIN {X -0.069,Y -597.719,Z 1441.005,A 0.000,B 0.000,C 90.000,E1 36.996} C_DIS
LIN {X 0.029,Y -595.761,Z 1441.000,A 0.000,B 0.000,C 90.000,E1 35.931} C_DIS
LIN {X -0.124,Y -594.086,Z 1440.995,A 0.000,B 0.000,C 90.000,E1 35.152} C_DIS
LIN {X 0.283,Y -590.893,Z 1440.988,A 0.000,B 0.000,C 90.000,E1 33.785} C_DIS
LIN {X -0.049,Y -587.967,Z 1440.982,A 0.000,B 0.000,C 90.000,E1 32.752} C_DIS
LIN {X 0.074,Y -584.668,Z 1440.976,A 0.000,B 0.000,C 90.000,E1 31.671} C_DIS
LIN {X 0.116,Y -582.786,Z 1440.973,A 0.000,B 0.000,C 90.000,E1 31.131} C_DIS
LIN {X 0.144,Y -580.700,Z 1440.970,A 0.000,B 0.000,C 90.000,E1 30.590} C_DIS
LIN {X -0.133,Y -578.418,Z 1440.967,A 0.000,B 0.000,C 90.000,E1 30.079} C_DIS
LIN {X -0.082,Y -574.022,Z 1440.962,A 0.000,B 0.000,C 90.000,E1 29.127} C_DIS
LIN {X -0.064,Y -569.827,Z 1440.957,A 0.000,B 0.000,C 90.000,E1 28.309} C_DIS
LIN {X -0.138,Y -566.799,Z 1440.954,A 0.000,B 0.000,C 90.000,E1 27.769} C_DIS
LIN {X -0.025,Y -561.159,Z 1440.949,A 0.000,B 0.000,C 90.000,E1 26.796} C_DIS
LIN {X -0.234,Y -555.049,Z 1440.943,A 0.000,B 0.000,C 90.000,E1 25.848} C_DIS
LIN {X -0.281,Y -550.353,Z 1440.940,A 0.000,B 0.000,C 90.000,E1 25.155} C_DIS
LIN {X 0.354,Y -545.154,Z 1440.936,A 0.000,B 0.000,C 90.000,E1 24.387} C_DIS
LIN {X -0.020,Y -541.882,Z 1440.933,A 0.000,B 0.000,C 90.000,E1 24.003} C_DIS
LIN {X 0.303,Y -536.042,Z 1440.929,A 0.000,B 0.000,C 90.000,E1 23.259} C_DIS
LIN {X -0.263,Y -528.660,Z 1440.925,A 0.000,B 0.000,C 90.000,E1 22.461} C_DIS
LIN {X -0.162,Y -519.749,Z 1440.919,A 0.000,B 0.000,C 90.000,E1 21.461} C_DIS
LIN {X 0.049,Y -509.046,Z 1440.913,A 0.000,B 0.000,C 90.000,E1 20.301} C_DIS
LIN {X 0.005,Y -499.603,Z 1440.907,A 0.000,B 0.000,C 90.000,E1 19.322} C_DIS
LIN {X 0.183,Y -487.313,Z 1440.901,A 0.000,B 0.000,C 90.000,E1 18.055} C_DIS
LIN {X 0.112,Y -472.654,Z 1440.892,A 0.000,B 0.000,C 90.000,E1 16.496} C_DIS
LIN {X -0.066,Y -460.769,Z 1440.884,A 0.000,B 0.000,C 90.000,E1 15.190} C_DIS
LIN {X -0.103,Y -455.014,Z 1440.881,A 0.000,B 0.000,C 90.000,E1 14.592} C_DIS
LIN {X 0.224,Y -450.450,Z 1440.879,A 0.000,B 0.000,C 90.000,E1 14.120} C_DIS
LIN {X -0.199,Y -445.409,Z 1440.876,A 0.000,B 0.000,C 90.000,E1 13.772} C_DIS
LIN {X -0.211,Y -441.631,Z 1440.875,A 0.000,B 0.000,C 90.000,E1 13.536} C_DIS
LIN {X -0.196,Y -439.022,Z 1440.874,A 0.000,B 0.000,C 90.000,E1 13.411} C_DIS
LIN {X -0.130,Y -437.432,Z 1440.874,A 0.000,B 0.000,C 90.000,E1 13.355} C_DIS
LIN {X 0.192,Y -436.253,Z 1440.874,A 0.000,B 0.000,C 90.000,E1 13.300} C_DIS
LIN {X 0.141,Y -368.853,Z 1440.874,A 0.000,B 0.000,C 90.000,E1 13.300} C_DIS
LIN {X -0.066,Y -366.364,Z 1440.854,A 0.000,B 0.000,C 90.000,E1 9.792} C_DIS
LIN {X -0.127,Y -361.725,Z 1440.821,A 0.000,B 0.000,C 90.000,E1 3.841} C_DIS
LIN {X 0.120,Y -360.842,Z 1440.800,A 0.000,B 0.000,C 90.000,E1 0.057} C_DIS
LIN {X -0.053,Y -359.426,Z 1440.770,A 0.000,B 0.000,C 90.000,E1 354.546} C_DIS
LIN {X 0.070,Y -358.890,Z 1440.759,A 0.000,B 0.000,C 90.000,E1 352.648} C_DIS
LIN {X -0.020,Y -359.563,Z 1440.726,A 0.000,B 0.000,C 90.000,E1 346.645} C_DIS
LIN {X 0.001,Y -361.801,Z 1440.684,A 0.000,B 0.000,C 90.000,E1 339.135} C_DIS
LIN {X -0.154,Y -362.053,Z 1440.680,A 0.000,B 0.000,C 90.000,E1 338.411} C_DIS
LIN {X 0.189,Y -365.980,Z 1440.643,A 0.000,B 0.000,C 90.000,E1 331.641} C_DIS
LIN {X 0.029,Y -366.387,Z 1440.639,A 0.000,B 0.000,C 90.000,E1 330.923} C_DIS
LIN {X -0.031,Y -371.355,Z 1440.604,A 0.000,B 0.000,C 90.000,E1 324.642} C_DIS
LIN {X -0.043,Y -371.766,Z 1440.602,A 0.000,B 0.000,C 90.000,E1 324.276} C_DIS
LIN {X 0.013,Y -377.358,Z 1440.567,A 0.000,B 0.000,C 90.000,E1 318.038} C_DIS
LIN {X 0.012,Y -378.235,Z 1440.563,A 0.000,B 0.000,C 90.000,E1 317.310} C_DIS
LIN {X 0.002,Y -383.940,Z 1440.531,A 0.000,B 0.000,C 90.000,E1 311.515} C_DIS
LIN {X 0.088,Y -384.893,Z 1440.527,A 0.000,B 0.000,C 90.000,E1 310.782} C_DIS
LIN {X 0.262,Y -390.610,Z 1440.495,A 0.000,B 0.000,C 90.000,E1 305.025} C_DIS
LIN {X 0.106,Y -391.104,Z 1440.493,A 0.000,B 0.000,C 90.000,E1 304.692} C_DIS
LIN {X 0.022,Y -391.648,Z 1440.489,A 0.000,B 0.000,C 90.000,E1 303.992} C_DIS
LIN {X -0.080,Y -396.825,Z 1440.459,A 0.000,B 0.000,C 90.000,E1 298.693} C_DIS
LIN {X -0.210,Y -397.120,Z 1440.457,A 0.000,B 0.000,C 90.000,E1 298.359} C_DIS
LIN {X -0.055,Y -401.597,Z 1440.426,A 0.000,B 0.000,C 90.000,E1 292.717} C_DIS
LIN {X 0.222,Y -404.659,Z 1440.395,A 0.000,B 0.000,C 90.000,E1 287.094} C_DIS
LIN {X -0.079,Y -404.735,Z 1440.391,A 0.000,B 0.000,C 90.000,E1 286.441} C_DIS
LIN {X 0.214,Y -406.099,Z 1440.364,A 0.000,B 0.000,C 90.000,E1 281.535} C_DIS
LIN {X -0.176,Y -406.094,Z 1440.362,A 0.000,B 0.000,C 90.000,E1 281.243} C_DIS
LIN {X -0.097,Y -405.680,Z 1440.333,A 0.000,B 0.000,C 90.000,E1 276.024} C_DIS
LIN {X -0.165,Y -405.058,Z 1440.328,A 0.000,B 0.000,C 90.000,E1 274.992} C_DIS
LIN {X -0.060,Y -403.497,Z 1440.304,A 0.000,B 0.000,C 90.000,E1 270.802} C_DIS
LIN {X -0.092,Y -403.288,Z 1440.302,A 0.000,B 0.000,C 90.000,E1 270.458} C_DIS
LIN {X 0.091,Y -398.931,Z 1440.271,A 0.000,B 0.000,C 90.000,E1 264.837} C_DIS
LIN {X -0.040,Y -393.108,Z 1440.242,A 0.000,B 0.000,C 90.000,E1 259.567} C_DIS
LIN {X -0.079,Y -392.835,Z 1440.240,A 0.000,B 0.000,C 90.000,E1 259.218} C_DIS
LIN {X 0.034,Y -385.993,Z 1440.212,A 0.000,B 0.000,C 90.000,E1 254.212} C_DIS
LIN {X -0.026,Y -385.267,Z 1440.208,A 0.000,B 0.000,C 90.000,E1 253.504} C_DIS
LIN {X -0.004,Y -384.768,Z 1440.206,A 0.000,B 0.000,C 90.000,E1 253.142} C_DIS
LIN {X 0.221,Y -377.973,Z 1440.182,A 0.000,B 0.000,C 90.000,E1 248.773} C_DIS
LIN {X -0.044,Y -376.233,Z 1440.174,A 0.000,B 0.000,C 90.000,E1 247.358} C_DIS
LIN {X 0.057,Y -374.944,Z 1440.170,A 0.000,B 0.000,C 90.000,E1 246.613} C_DIS
LIN {X -0.208,Y -368.417,Z 1440.148,A 0.000,B 0.000,C 90.000,E1 242.615} C_DIS
LIN {X 0.097,Y -366.047,Z 1440.137,A 0.000,B 0.000,C 90.000,E1 240.717} C_DIS
LIN {X 0.004,Y -359.196,Z 1440.115,A 0.000,B 0.000,C 90.000,E1 236.628} C_DIS
LIN {X 0.021,Y -355.842,Z 1440.100,A 0.000,B 0.000,C 90.000,E1 233.989} C_DIS
LIN {X -0.173,Y -348.793,Z 1440.075,A 0.000,B 0.000,C 90.000,E1 229.461} C_DIS
LIN {X -0.097,Y -346.185,Z 1440.062,A 0.000,B 0.000,C 90.000,E1 227.148} C_DIS
LIN {X -0.088,Y -345.065,Z 1440.058,A 0.000,B 0.000,C 90.000,E1 226.377} C_DIS
LIN {X 0.094,Y -338.586,Z 1440.030,A 0.000,B 0.000,C 90.000,E1 221.310} C_DIS
LIN {X 0.094,Y -336.840,Z 1440.019,A 0.000,B 0.000,C 90.000,E1 219.358} C_DIS
LIN {X 0.014,Y -330.861,Z 1439.988,A 0.000,B 0.000,C 90.000,E1 213.865} C_DIS
LIN {X 0.149,Y -329.296,Z 1439.975,A 0.000,B 0.000,C 90.000,E1 211.465} C_DIS
LIN {X -0.154,Y -324.669,Z 1439.942,A 0.000,B 0.000,C 90.000,E1 205.540} C_DIS
LIN {X 0.174,Y -323.837,Z 1439.928,A 0.000,B 0.000,C 90.000,E1 203.078} C_DIS
LIN {X -0.017,Y -321.124,Z 1439.881,A 0.000,B 0.000,C 90.000,E1 194.662} C_DIS
LIN {X 0.138,Y -320.932,Z 1439.877,A 0.000,B 0.000,C 90.000,E1 193.828} C_DIS
LIN {X -0.076,Y -321.562,Z 1439.832,A 0.000,B 0.000,C 90.000,E1 185.796} C_DIS
LIN {X -0.143,Y -324.415,Z 1439.790,A 0.000,B 0.000,C 90.000,E1 178.165} C_DIS
LIN {X -0.141,Y -325.376,Z 1439.783,A 0.000,B 0.000,C 90.000,E1 176.963} C_DIS
LIN {X -0.100,Y -329.112,Z 1439.750,A 0.000,B 0.000,C 90.000,E1 170.971} C_DIS
LIN {X 0.061,Y -334.260,Z 1439.726,A 0.000,B 0.000,C 90.000,E1 166.589} C_DIS
LIN {X 0.016,Y -335.626,Z 1439.718,A 0.000,B 0.000,C 90.000,E1 165.283} C_DIS
LIN {X 0.030,Y -335.871,Z 1439.717,A 0.000,B 0.000,C 90.000,E1 165.046} C_DIS
LIN {X 0.010,Y -374.949,Z 1439.717,A 0.000,B 0.000,C 90.000,E1 165.046} C_DIS
LIN {X -0.128,Y -376.207,Z 1439.717,A 0.000,B 0.000,C 90.000,E1 165.046} C_DIS
LIN {X 0.154,Y -378.318,Z 1439.716,A 0.000,B 0.000,C 90.000,E1 164.936} C_DIS
LIN {X -0.149,Y -380.852,Z 1439.716,A 0.000,B 0.000,C 90.000,E1 164.866} C_DIS
LIN {X -0.021,Y -383.735,Z 1439.715,A 0.000,B 0.000,C 90.000,E1 164.685} C_DIS
LIN {X -0.208,Y -386.755,Z 1439.714,A 0.000,B 0.000,C 90.000,E1 164.519} C_DIS
LIN {X 0.033,Y -392.929,Z 1439.711,A 0.000,B 0.000,C 90.000,E1 164.031} C_DIS
LIN {X 0.172,Y -399.229,Z 1439.708,A 0.000,B 0.000,C 90.000,E1 163.504} C_DIS
LIN {X -0.098,Y -408.544,Z 1439.704,A 0.000,B 0.000,C 90.000,E1 162.725} C_DIS
LIN {X -0.058,Y -425.573,Z 1439.696,A 0.000,B 0.000,C 90.000,E1 161.221} C_DIS
LIN {X 0.082,Y -439.522,Z 1439.689,A 0.000,B 0.000,C 90.000,E1 160.007} C_DIS
LIN {X -0.016,Y -453.420,Z 1439.682,A 0.000,B 0.000,C 90.000,E1 158.847} C_DIS
LIN {X -0.092,Y -463.890,Z 1439.678,A 0.000,B 0.000,C 90.000,E1 157.975} C_DIS
LIN {X 0.083,Y -474.451,Z 1439.673,A 0.000,B 0.000,C 90.000,E1 157.050} C_DIS
LIN {X -0.274,Y -484.772,Z 1439.667,A 0.000,B 0.000,C 90.000,E1 156.177} C_DIS
LIN {X -0.158,Y -493.365,Z 1439.663,A 0.000,B 0.000,C 90.000,E1 155.357} C_DIS
LIN {X -0.125,Y -501.638,Z 1439.658,A 0.000,B 0.000,C 90.000,E1 154.537} C_DIS
LIN {X 0.069,Y -506.992,Z 1439.655,A 0.000,B 0.000,C 90.000,E1 153.948} C_DIS
LIN {X 0.079,Y -510.885,Z 1439.653,A 0.000,B 0.000,C 90.000,E1 153.512} C_DIS
LIN {X 0.102,Y -515.640,Z 1439.650,A 0.000,B 0.000,C 90.000,E1 152.922} C_DIS
LIN {X -0.122,Y -520.036,Z 1439.646,A 0.000,B 0.000,C 90.000,E1 152.359} C_DIS
LIN {X 0.087,Y -523.074,Z 1439.644,A 0.000,B 0.000,C 90.000,E1 151.897} C_DIS
LIN {X 0.004,Y -527.457,Z 1439.640,A 0.000,B 0.000,C 90.000,E1 151.179} C_DIS
LIN {X 0.109,Y -530.571,Z 1439.637,A 0.000,B 0.000,C 90.000,E1 150.589} C_DIS
LIN {X 0.089,Y -534.036,Z 1439.633,A 0.000,B 0.000,C 90.000,E1 149.871} C_DIS
LIN {X -0.220,Y -536.490,Z 1439.630,A 0.000,B 0.000,C 90.000,E1 149.331} C_DIS
LIN {X -0.054,Y -538.752,Z 1439.626,A 0.000,B 0.000,C 90.000,E1 148.742} C_DIS
LIN {X 0.133,Y -541.631,Z 1439.622,A 0.000,B 0.000,C 90.000,E1 147.867} C_DIS
LIN {X -0.128,Y -543.404,Z 1439.618,A 0.000,B 0.000,C 90.000,E1 147.327} C_DIS
LIN {X 0.137,Y -546.480,Z 1439.612,A 0.000,B 0.000,C 90.000,E1 146.167} C_DIS
LIN {X 0.258,Y -548.567,Z 1439.607,A 0.000,B 0.000,C 90.000,E1 145.308} C_DIS
LIN {X 0.093,Y -550.370,Z 1439.603,A 0.000,B 0.000,C 90.000,E1 144.482} C_DIS
LIN {X 0.265,Y -551.899,Z 1439.598,A 0.000,B 0.000,C 90.000,E1 143.623} C_DIS
LIN {X -0.319,Y -553.216,Z 1439.593,A 0.000,B 0.000,C 90.000,E1 142.844} C_DIS
LIN {X -0.047,Y -554.707,Z 1439.587,A 0.000,B 0.000,C 90.000,E1 141.698} C_DIS
LIN {X -0.266,Y -555.670,Z 1439.583,A 0.000,B 0.000,C 90.000,E1 140.884} C_DIS
LIN {X 0.034,Y -556.977,Z 1439.575,A 0.000,B 0.000,C 90.000,E1 139.461} C_DIS
LIN {X 0.010,Y -558.299,Z 1439.566,A 0.000,B 0.000,C 90.000,E1 137.796} C_DIS
LIN {X 0.310,Y -559.318,Z 1439.558,A 0.000,B 0.000,C 90.000,E1 136.377} C_DIS
LIN {X -0.232,Y -559.937,Z 1439.552,A 0.000,B 0.000,C 90.000,E1 135.324} C_DIS
LIN {X -0.301,Y -560.518,Z 1439.544,A 0.000,B 0.000,C 90.000,E1 133.947} C_DIS
LIN {X 0.039,Y -560.953,Z 1439.536,A 0.000,B 0.000,C 90.000,E1 132.528} C_DIS
LIN {X -0.079,Y -561.076,Z 1439.530,A 0.000,B 0.000,C 90.000,E1 131.434} C_DIS
LIN {X -0.025,Y -561.157,Z 1439.521,A 0.000,B 0.000,C 90.000,E1 129.769} C_DIS
LIN {X 0.013,Y -561.235,Z 1439.513,A 0.000,B 0.000,C 90.000,E1 128.382} C_DIS
LIN {X 0.051,Y -561.176,Z 1439.506,A 0.000,B 0.000,C 90.000,E1 126.996} C_DIS
LIN {X 0.106,Y -561.094,Z 1439.500,A 0.000,B 0.000,C 90.000,E1 125.884} C_DIS
LIN {X -0.103,Y -560.873,Z 1439.490,A 0.000,B 0.000,C 90.000,E1 124.246} C_DIS
LIN {X 0.201,Y -560.581,Z 1439.483,A 0.000,B 0.000,C 90.000,E1 122.832} C_DIS
LIN {X -0.081,Y -560.416,Z 1439.464,A 0.000,B 0.000,C 90.000,E1 119.539} C_DIS
LIN {X -0.173,Y -560.973,Z 1439.452,A 0.000,B 0.000,C 90.000,E1 117.334} C_DIS
LIN {X -0.105,Y -561.565,Z 1439.443,A 0.000,B 0.000,C 90.000,E1 115.668} C_DIS
LIN {X 0.159,Y -562.023,Z 1439.435,A 0.000,B 0.000,C 90.000,E1 114.259} C_DIS
LIN {X -0.031,Y -562.385,Z 1439.427,A 0.000,B 0.000,C 90.000,E1 112.898} C_DIS
LIN {X 0.228,Y -563.394,Z 1439.415,A 0.000,B 0.000,C 90.000,E1 110.663} C_DIS
LIN {X 0.145,Y -564.092,Z 1439.412,A 0.000,B 0.000,C 90.000,E1 110.120} C_DIS
LIN {X 0.217,Y -564.443,Z 1439.409,A 0.000,B 0.000,C 90.000,E1 109.631} C_DIS
LIN {X -0.252,Y -565.996,Z 1439.407,A 0.000,B 0.000,C 90.000,E1 109.268} C_DIS
LIN {X 0.324,Y -566.407,Z 1439.407,A 0.000,B 0.000,C 90.000,E1 109.141} C_DIS
LIN {X -0.211,Y -569.277,Z 1439.405,A 0.000,B 0.000,C 90.000,E1 108.852} C_DIS
LIN {X -0.096,Y -576.289,Z 1439.402,A 0.000,B 0.000,C 90.000,E1 108.362} C_DIS
LIN {X -0.290,Y -579.335,Z 1439.401,A 0.000,B 0.000,C 90.000,E1 108.181} C_DIS
LIN {X 0.255,Y -583.549,Z 1439.399,A 0.000,B 0.000,C 90.000,E1 107.819} C_DIS
LIN {X -0.151,Y -586.062,Z 1439.398,A 0.000,B 0.000,C 90.000,E1 107.638} C_DIS
LIN {X -0.196,Y -589.900,Z 1439.396,A 0.000,B 0.000,C 90.000,E1 107.275} C_DIS
LIN {X 0.090,Y -594.564,Z 1439.393,A 0.000,B 0.000,C 90.000,E1 106.732} C_DIS
LIN {X -0.003,Y -599.432,Z 1439.389,A 0.000,B 0.000,C 90.000,E1 106.079} C_DIS
LIN {X -0.056,Y -602.847,Z 1439.386,A 0.000,B 0.000,C 90.000,E1 105.426} C_DIS
LIN {X 0.250,Y -603.894,Z 1439.384,A 0.000,B 0.000,C 90.000,E1 105.134} C_DIS
LIN {X -0.141,Y -605.283,Z 1439.381,A 0.000,B 0.000,C 90.000,E1 104.647} C_DIS
LIN {X -0.091,Y -606.434,Z 1439.378,A 0.000,B 0.000,C 90.000,E1 104.120} C_DIS
LIN {X -0.031,Y -607.261,Z 1439.375,A 0.000,B 0.000,C 90.000,E1 103.592} C_DIS
LIN {X -0.222,Y -608.096,Z 1439.371,A 0.000,B 0.000,C 90.000,E1 102.827} C_DIS
LIN {X 0.189,Y -608.572,Z 1439.367,A 0.000,B 0.000,C 90.000,E1 102.007} C_DIS
LIN {X 0.269,Y -608.607,Z 1439.364,A 0.000,B 0.000,C 90.000,E1 101.478} C_DIS
LIN {X -0.251,Y -608.078,Z 1439.361,A 0.000,B 0.000,C 90.000,E1 101.007} C_DIS
LIN {X -0.290,Y -607.277,Z 1439.358,A 0.000,B 0.000,C 90.000,E1 100.489} C_DIS
LIN {X -0.222,Y -606.161,Z 1439.355,A 0.000,B 0.000,C 90.000,E1 99.962} C_DIS
LIN {X 0.106,Y -605.511,Z 1439.354,A 0.000,B 0.000,C 90.000,E1 99.670} C_DIS
LIN {X 0.059,Y -603.949,Z 1439.351,A 0.000,B 0.000,C 90.000,E1 99.151} C_DIS
LIN {X 0.098,Y -601.889,Z 1439.348,A 0.000,B 0.000,C 90.000,E1 98.624} C_DIS
LIN {X -0.266,Y -597.966,Z 1439.344,A 0.000,B 0.000,C 90.000,E1 97.871} C_DIS
LIN {X -0.155,Y -593.612,Z 1439.339,A 0.000,B 0.000,C 90.000,E1 97.068} C_DIS
LIN {X -0.205,Y -590.173,Z 1439.336,A 0.000,B 0.000,C 90.000,E1 96.543} C_DIS
LIN {X -0.014,Y -588.318,Z 1439.335,A 0.000,B 0.000,C 90.000,E1 96.258} C_DIS
LIN {X 0.233,Y -586.230,Z 1439.333,A 0.000,B 0.000,C 90.000,E1 95.967} C_DIS
LIN {X -0.170,Y -583.793,Z 1439.332,A 0.000,B 0.000,C 90.000,E1 95.739} C_DIS
LIN {X -0.236,Y -574.610,Z 1439.327,A 0.000,B 0.000,C 90.000,E1 94.878} C_DIS
LIN {X 0.254,Y -573.542,Z 1439.326,A 0.000,B 0.000,C 90.000,E1 94.702} C_DIS
LIN {X -0.071,Y -571.917,Z 1439.325,A 0.000,B 0.000,C 90.000,E1 94.473} C_DIS
LIN {X 0.066,Y -571.057,Z 1439.323,A 0.000,B 0.000,C 90.000,E1 94.188} C_DIS
LIN {X 0.235,Y -570.631,Z 1439.322,A 0.000,B 0.000,C 90.000,E1 93.898} C_DIS
LIN {X -0.080,Y -570.482,Z 1439.319,A 0.000,B 0.000,C 90.000,E1 93.383} C_DIS
LIN {X 0.158,Y -572.426,Z 1439.304,A 0.000,B 0.000,C 90.000,E1 90.630} C_DIS
LIN {X -0.287,Y -573.661,Z 1439.296,A 0.000,B 0.000,C 90.000,E1 89.312} C_DIS
LIN {X 0.169,Y -575.405,Z 1439.286,A 0.000,B 0.000,C 90.000,E1 87.364} C_DIS
LIN {X -0.028,Y -576.908,Z 1439.276,A 0.000,B 0.000,C 90.000,E1 85.755} C_DIS
LIN {X 0.233,Y -578.196,Z 1439.269,A 0.000,B 0.000,C 90.000,E1 84.375} C_DIS
LIN {X -0.069,Y -580.323,Z 1439.257,A 0.000,B 0.000,C 90.000,E1 82.243} C_DIS
LIN {X -0.181,Y -581.701,Z 1439.249,A 0.000,B 0.000,C 90.000,E1 80.905} C_DIS
LIN {X 0.104,Y -583.554,Z 1439.239,A 0.000,B 0.000,C 90.000,E1 78.993} C_DIS
LIN {X -0.083,Y -584.685,Z 1439.233,A 0.000,B 0.000,C 90.000,E1 77.937} C_DIS
LIN {X 0.074,Y -585.433,Z 1439.229,A 0.000,B 0.000,C 90.000,E1 77.117} C_DIS
LIN {X -0.023,Y -586.671,Z 1439.220,A 0.000,B 0.000,C 90.000,E1 75.519} C_DIS
LIN {X -0.019,Y -587.427,Z 1439.214,A 0.000,B 0.000,C 90.000,E1 74.448} C_DIS
LIN {X 0.090,Y -588.366,Z 1439.205,A 0.000,B 0.000,C 90.000,E1 72.834} C_DIS
LIN {X 0.108,Y -588.990,Z 1439.199,A 0.000,B 0.000,C 90.000,E1 71.764} C_DIS
LIN {X 0.286,Y -589.931,Z 1439.188,A 0.000,B 0.000,C 90.000,E1 69.880} C_DIS
LIN {X -0.184,Y -591.137,Z 1439.177,A 0.000,B 0.000,C 90.000,E1 67.794} C_DIS
LIN {X 0.034,Y -592.005,Z 1439.168,A 0.000,B 0.000,C 90.000,E1 66.177} C_DIS
LIN {X 0.224,Y -593.665,Z 1439.154,A 0.000,B 0.000,C 90.000,E1 63.768} C_DIS
LIN {X -0.057,Y -594.357,Z 1439.150,A 0.000,B 0.000,C 90.000,E1 62.999} C_DIS
LIN {X 0.040,Y -596.648,Z 1439.134,A 0.000,B 0.000,C 90.000,E1 60.078} C_DIS
LIN {X -0.180,Y -598.289,Z 1439.124,A 0.000,B 0.000,C 90.000,E1 58.250} C_DIS
LIN {X 0.098,Y -599.239,Z 1439.118,A 0.000,B 0.000,C 90.000,E1 57.168} C_DIS
LIN {X -0.209,Y -600.416,Z 1439.110,A 0.000,B 0.000,C 90.000,E1 55.881} C_DIS
LIN {X -0.067,Y -601.351,Z 1439.104,A 0.000,B 0.000,C 90.000,E1 54.815} C_DIS
LIN {X -0.009,Y -602.409,Z 1439.097,A 0.000,B 0.000,C 90.000,E1 53.497} C_DIS
LIN {X 0.192,Y -603.572,Z 1439.089,A 0.000,B 0.000,C 90.000,E1 51.904} C_DIS
LIN {X 0.154,Y -604.360,Z 1439.081,A 0.000,B 0.000,C 90.000,E1 50.598} C_DIS
LIN {X 0.252,Y -604.911,Z 1439.075,A 0.000,B 0.000,C 90.000,E1 49.542} C_DIS
LIN {X 0.159,Y -605.165,Z 1439.068,A 0.000,B 0.000,C 90.000,E1 48.243} C_DIS
LIN {X -0.131,Y -605.420,Z 1439.059,A 0.000,B 0.000,C 90.000,E1 46.701} C_DIS
LIN {X -0.009,Y -605.483,Z 1439.051,A 0.000,B 0.000,C 90.000,E1 45.121} C_DIS
LIN {X -0.355,Y -605.125,Z 1439.045,A 0.000,B 0.000,C 90.000,E1 44.109} C_DIS
LIN {X 0.159,Y -604.580,Z 1439.039,A 0.000,B 0.000,C 90.000,E1 43.014} C_DIS
LIN {X -0.187,Y -603.886,Z 1439.033,A 0.000,B 0.000,C 90.000,E1 42.000} C_DIS
LIN {X -0.343,Y -603.255,Z 1439.029,A 0.000,B 0.000,C 90.000,E1 41.229} C_DIS
LIN {X -0.007,Y -601.881,Z 1439.022,A 0.000,B 0.000,C 90.000,E1 39.886} C_DIS
LIN {X -0.167,Y -600.281,Z 1439.014,A 0.000,B 0.000,C 90.000,E1 38.588} C_DIS
LIN {X 0.205,Y -598.379,Z 1439.007,A 0.000,B 0.000,C 90.000,E1 37.237} C_DIS
LIN {X -0.163,Y -596.476,Z 1439.001,A 0.000,B 0.000,C 90.000,E1 36.217} C_DIS
LIN {X 0.178,Y -594.876,Z 1438.997,A 0.000,B 0.000,C 90.000,E1 35.391} C_DIS
LIN {X 0.236,Y -592.451,Z 1438.991,A 0.000,B 0.000,C 90.000,E1 34.326} C_DIS
LIN {X -0.282,Y -590.439,Z 1438.986,A 0.000,B 0.000,C 90.000,E1 33.579} C_DIS
LIN {X 0.193,Y -587.452,Z 1438.980,A 0.000,B 0.000,C 90.000,E1 32.467} C_DIS
LIN {X 0.126,Y -584.999,Z 1438.976,A 0.000,B 0.000,C 90.000,E1 31.671} C_DIS
LIN {X -0.002,Y -584.133,Z 1438.975,A 0.000,B 0.000,C 90.000,E1 31.416} C_DIS
LIN {X 0.201,Y -581.056,Z 1438.970,A 0.000,B 0.000,C 90.000,E1 30.590} C_DIS
LIN {X 0.071,Y -577.586,Z 1438.966,A 0.000,B 0.000,C 90.000,E1 29.795} C_DIS
LIN {X -0.097,Y -573.781,Z 1438.961,A 0.000,B 0.000,C 90.000,E1 28.999} C_DIS
LIN {X 0.004,Y -570.274,Z 1438.957,A 0.000,B 0.000,C 90.000,E1 28.309} C_DIS
LIN {X -0.069,Y -567.264,Z 1438.954,A 0.000,B 0.000,C 90.000,E1 27.769} C_DIS
LIN {X 0.050,Y -561.619,Z 1438.949,A 0.000,B 0.000,C 90.000,E1 26.796} C_DIS
LIN {X -0.155,Y -555.517,Z 1438.944,A 0.000,B 0.000,C 90.000,E1 25.848} C_DIS
LIN {X -0.198,Y -550.904,Z 1438.940,A 0.000,B 0.000,C 90.000,E1 25.155} C_DIS
LIN {X -0.160,Y -546.840,Z 1438.937,A 0.000,B 0.000,C 90.000,E1 24.591} C_DIS
LIN {X -0.278,Y -541.343,Z 1438.933,A 0.000,B 0.000,C 90.000,E1 23.898} C_DIS
LIN {X 0.168,Y -535.593,Z 1438.929,A 0.000,B 0.000,C 90.000,E1 23.153} C_DIS
LIN {X -0.119,Y -528.207,Z 1438.924,A 0.000,B 0.000,C 90.000,E1 22.333} C_DIS
LIN {X 0.150,Y -520.604,Z 1438.919,A 0.000,B 0.000,C 90.000,E1 21.461} C_DIS
LIN {X -0.201,Y -513.953,Z 1438.915,A 0.000,B 0.000,C 90.000,E1 20.791} C_DIS
LIN {X -0.167,Y -505.870,Z 1438.911,A 0.000,B 0.000,C 90.000,E1 19.939} C_DIS
LIN {X 0.040,Y -499.089,Z 1438.907,A 0.000,B 0.000,C 90.000,E1 19.214} C_DIS
LIN {X -0.178,Y -488.209,Z 1438.901,A 0.000,B 0.000,C 90.000,E1 18.127} C_DIS
LIN {X -0.038,Y -472.024,Z 1438.891,A 0.000,B 0.000,C 90.000,E1 16.386} C_DIS
LIN {X 0.152,Y -457.397,Z 1438.882,A 0.000,B 0.000,C 90.000,E1 14.717} C_DIS
LIN {X -0.027,Y -451.821,Z 1438.878,A 0.000,B 0.000,C 90.000,E1 14.120} C_DIS
LIN {X 0.167,Y -447.265,Z 1438.876,A 0.000,B 0.000,C 90.000,E1 13.647} C_DIS
LIN {X 0.100,Y -442.502,Z 1438.874,A 0.000,B 0.000,C 90.000,E1 13.244} C_DIS
LIN {X -0.050,Y -439.165,Z 1438.872,A 0.000,B 0.000,C 90.000,E1 13.008} C_DIS
LIN {X -0.030,Y -435.384,Z 1438.871,A 0.000,B 0.000,C 90.000,E1 12.771} C_DIS
LIN {X 0.087,Y -432.854,Z 1438.870,A 0.000,B 0.000,C 90.000,E1 12.647} C_DIS
LIN {X 0.216,Y -430.847,Z 1438.870,A 0.000,B 0.000,C 90.000,E1 12.591} C_DIS
LIN {X 0.161,Y -368.249,Z 1438.870,A 0.000,B 0.000,C 90.000,E1 12.591} C_DIS
LIN {X 0.064,Y -366.482,Z 1438.855,A 0.000,B 0.000,C 90.000,E1 9.905} C_DIS
LIN {X 0.000,Y -361.785,Z 1438.822,A 0.000,B 0.000,C 90.000,E1 3.955} C_DIS
LIN {X -0.114,Y -360.900,Z 1438.801,A 0.000,B 0.000,C 90.000,E1 0.229} C_DIS
LIN {X -0.053,Y -359.426,Z 1438.770,A 0.000,B 0.000,C 90.000,E1 354.546} C_DIS
LIN {X 0.070,Y -358.890,Z 1438.759,A 0.000,B 0.000,C 90.000,E1 352.648} C_DIS
LIN {X -0.020,Y -359.563,Z 1438.726,A 0.000,B 0.000,C 90.000,E1 346.645} C_DIS
LIN {X 0.001,Y -361.801,Z 1438.684,A 0.000,B 0.000,C 90.000,E1 339.135} C_DIS
LIN {X -0.154,Y -362.053,Z 1438.680,A 0.000,B 0.000,C 90.000,E1 338.411} C_DIS
LIN {X 0.189,Y -365.980,Z 1438.643,A 0.000,B 0.000,C 90.000,E1 331.641} C_DIS
LIN {X 0.029,Y -366.387,Z 1438.639,A 0.000,B 0.000,C 90.000,E1 330.923} C_DIS
LIN {X -0.031,Y -371.355,Z 1438.604,A 0.000,B 0.000,C 90.000,E1 324.642} C_DIS
LIN {X -0.043,Y -371.766,Z 1438.602,A 0.000,B 0.000,C 90.000,E1 324.276} C_DIS
LIN {X 0.013,Y -377.358,Z 1438.567,A 0.000,B 0.000,C 90.000,E1 318.038} C_DIS
LIN {X 0.012,Y -378.235,Z 1438.563,A 0.000,B 0.000,C 90.000,E1 317.310} C_DIS
LIN {X 0.002,Y -383.940,Z 1438.531,A 0.000,B 0.000,C 90.000,E1 311.515} C_DIS
LIN {X 0.088,Y -384.893,Z 1438.527,A 0.000,B 0.000,C 90.000,E1 310.782} C_DIS
LIN {X 0.262,Y -390.610,Z 1438.495,A 0.000,B 0.000,C 90.000,E1 305.025} C_DIS
LIN {X 0.106,Y -391.104,Z 1438.493,A 0.000,B 0.000,C 90.000,E1 304.692} C_DIS
LIN {X 0.022,Y -391.648,Z 1438.489,A 0.000,B 0.000,C 90.000,E1 303.992} C_DIS
LIN {X -0.080,Y -396.825,Z 1438.459,A 0.000,B 0.000,C 90.000,E1 298.693} C_DIS
LIN {X -0.210,Y -397.120,Z 1438.457,A 0.000,B 0.000,C 90.000,E1 298.359} C_DIS
LIN {X -0.055,Y -401.597,Z 1438.426,A 0.000,B 0.000,C 90.000,E1 292.717} C_DIS
LIN {X 0.222,Y -404.659,Z 1438.395,A 0.000,B 0.000,C 90.000,E1 287.094} C_DIS
LIN {X -0.079,Y -404.735,Z 1438.391,A 0.000,B 0.000,C 90.000,E1 286.441} C_DIS
LIN {X 0.214,Y -406.099,Z 1438.364,A 0.000,B 0.000,C 90.000,E1 281.535} C_DIS
LIN {X -0.176,Y -406.094,Z 1438.362,A 0.000,B 0.000,C 90.000,E1 281.243} C_DIS
LIN {X -0.097,Y -405.680,Z 1438.333,A 0.000,B 0.000,C 90.000,E1 276.024} C_DIS
LIN {X -0.165,Y -405.058,Z 1438.328,A 0.000,B 0.000,C 90.000,E1 274.992} C_DIS
LIN {X -0.060,Y -403.497,Z 1438.304,A 0.000,B 0.000,C 90.000,E1 270.802} C_DIS
LIN {X -0.092,Y -403.288,Z 1438.302,A 0.000,B 0.000,C 90.000,E1 270.458} C_DIS
LIN {X 0.091,Y -398.931,Z 1438.271,A 0.000,B 0.000,C 90.000,E1 264.837} C_DIS
LIN {X -0.040,Y -393.108,Z 1438.242,A 0.000,B 0.000,C 90.000,E1 259.567} C_DIS
LIN {X -0.079,Y -392.835,Z 1438.240,A 0.000,B 0.000,C 90.000,E1 259.218} C_DIS
LIN {X 0.034,Y -385.993,Z 1438.212,A 0.000,B 0.000,C 90.000,E1 254.212} C_DIS
LIN {X -0.026,Y -385.267,Z 1438.208,A 0.000,B 0.000,C 90.000,E1 253.504} C_DIS
LIN {X -0.004,Y -384.768,Z 1438.206,A 0.000,B 0.000,C 90.000,E1 253.142} C_DIS
LIN {X 0.221,Y -377.973,Z 1438.182,A 0.000,B 0.000,C 90.000,E1 248.773} C_DIS
LIN {X -0.044,Y -376.233,Z 1438.174,A 0.000,B 0.000,C 90.000,E1 247.358} C_DIS
LIN {X 0.057,Y -374.944,Z 1438.170,A 0.000,B 0.000,C 90.000,E1 246.613} C_DIS
LIN {X -0.208,Y -368.417,Z 1438.148,A 0.000,B 0.000,C 90.000,E1 242.615} C_DIS
LIN {X 0.097,Y -366.047,Z 1438.137,A 0.000,B 0.000,C 90.000,E1 240.717} C_DIS
LIN {X 0.004,Y -359.196,Z 1438.115,A 0.000,B 0.000,C 90.000,E1 236.628} C_DIS
LIN {X 0.021,Y -355.842,Z 1438.100,A 0.000,B 0.000,C 90.000,E1 233.989} C_DIS
LIN {X -0.173,Y -348.793,Z 1438.075,A 0.000,B 0.000,C 90.000,E1 229.461} C_DIS
LIN {X -0.097,Y -346.185,Z 1438.062,A 0.000,B 0.000,C 90.000,E1 227.148} C_DIS
LIN {X -0.088,Y -345.065,Z 1438.058,A 0.000,B 0.000,C 90.000,E1 226.377} C_DIS
LIN {X 0.094,Y -338.586,Z 1438.030,A 0.000,B 0.000,C 90.000,E1 221.310} C_DIS
LIN {X 0.094,Y -336.840,Z 1438.019,A 0.000,B 0.000,C 90.000,E1 219.358} C_DIS
LIN {X 0.014,Y -330.861,Z 1437.988,A 0.000,B 0.000,C 90.000,E1 213.865} C_DIS
LIN {X 0.149,Y -329.296,Z 1437.975,A 0.000,B 0.000,C 90.000,E1 211.465} C_DIS
LIN {X -0.154,Y -324.669,Z 1437.942,A 0.000,B 0.000,C 90.000,E1 205.540} C_DIS
LIN {X 0.174,Y -323.837,Z 1437.928,A 0.000,B 0.000,C 90.000,E1 203.078} C_DIS
LIN {X -0.017,Y -321.124,Z 1437.881,A 0.000,B 0.000,C 90.000,E1 194.662} C_DIS
LIN {X 0.138,Y -320.932,Z 1437.877,A 0.000,B 0.000,C 90.000,E1 193.828} C_DIS
LIN {X -0.076,Y -321.562,Z 1437.832,A 0.000,B 0.000,C 90.000,E1 185.796} C_DIS
LIN {X -0.143,Y -324.415,Z 1437.790,A 0.000,B 0.000,C 90.000,E1 178.165} C_DIS
LIN {X -0.141,Y -325.376,Z 1437.783,A 0.000,B 0.000,C 90.000,E1 176.963} C_DIS
LIN {X -0.100,Y -329.112,Z 1437.750,A 0.000,B 0.000,C 90.000,E1 170.971} C_DIS
LIN {X 0.061,Y -334.260,Z 1437.726,A 0.000,B 0.000,C 90.000,E1 166.589} C_DIS
LIN {X -0.015,Y -335.087,Z 1437.721,A 0.000,B 0.000,C 90.000,E1 165.825} C_DIS
LIN {X -0.048,Y -368.081,Z 1437.721,A 0.000,B 0.000,C 90.000,E1 165.825} C_DIS
LIN {X 0.108,Y -370.388,Z 1437.721,A 0.000,B 0.000,C 90.000,E1 165.755} C_DIS
LIN {X -0.103,Y -372.538,Z 1437.720,A 0.000,B 0.000,C 90.000,E1 165.700} C_DIS
LIN {X 0.124,Y -375.255,Z 1437.720,A 0.000,B 0.000,C 90.000,E1 165.519} C_DIS
LIN {X 0.084,Y -378.189,Z 1437.719,A 0.000,B 0.000,C 90.000,E1 165.338} C_DIS
LIN {X 0.207,Y -384.347,Z 1437.716,A 0.000,B 0.000,C 90.000,E1 164.866} C_DIS
LIN {X -0.103,Y -390.597,Z 1437.713,A 0.000,B 0.000,C 90.000,E1 164.393} C_DIS
LIN {X -0.107,Y -399.811,Z 1437.709,A 0.000,B 0.000,C 90.000,E1 163.559} C_DIS
LIN {X 0.109,Y -415.398,Z 1437.701,A 0.000,B 0.000,C 90.000,E1 162.127} C_DIS
LIN {X -0.152,Y -429.224,Z 1437.694,A 0.000,B 0.000,C 90.000,E1 160.967} C_DIS
LIN {X 0.068,Y -441.600,Z 1437.688,A 0.000,B 0.000,C 90.000,E1 159.880} C_DIS
LIN {X 0.127,Y -456.819,Z 1437.681,A 0.000,B 0.000,C 90.000,E1 158.592} C_DIS
LIN {X -0.066,Y -465.945,Z 1437.677,A 0.000,B 0.000,C 90.000,E1 157.847} C_DIS
LIN {X 0.149,Y -474.938,Z 1437.673,A 0.000,B 0.000,C 90.000,E1 157.050} C_DIS
LIN {X -0.201,Y -485.211,Z 1437.668,A 0.000,B 0.000,C 90.000,E1 156.177} C_DIS
LIN {X -0.077,Y -493.745,Z 1437.663,A 0.000,B 0.000,C 90.000,E1 155.357} C_DIS
LIN {X -0.076,Y -502.062,Z 1437.659,A 0.000,B 0.000,C 90.000,E1 154.537} C_DIS
LIN {X 0.003,Y -507.285,Z 1437.655,A 0.000,B 0.000,C 90.000,E1 153.973} C_DIS
LIN {X -0.157,Y -511.127,Z 1437.653,A 0.000,B 0.000,C 90.000,E1 153.563} C_DIS
LIN {X 0.093,Y -515.846,Z 1437.650,A 0.000,B 0.000,C 90.000,E1 152.948} C_DIS
LIN {X 0.108,Y -520.247,Z 1437.647,A 0.000,B 0.000,C 90.000,E1 152.359} C_DIS
LIN {X 0.157,Y -524.207,Z 1437.643,A 0.000,B 0.000,C 90.000,E1 151.769} C_DIS
LIN {X 0.239,Y -527.679,Z 1437.640,A 0.000,B 0.000,C 90.000,E1 151.179} C_DIS
LIN {X 0.196,Y -531.496,Z 1437.636,A 0.000,B 0.000,C 90.000,E1 150.461} C_DIS
LIN {X -0.131,Y -534.298,Z 1437.633,A 0.000,B 0.000,C 90.000,E1 149.921} C_DIS
LIN {X -0.260,Y -537.869,Z 1437.628,A 0.000,B 0.000,C 90.000,E1 149.076} C_DIS
LIN {X 0.195,Y -539.016,Z 1437.626,A 0.000,B 0.000,C 90.000,E1 148.742} C_DIS
LIN {X -0.350,Y -542.766,Z 1437.620,A 0.000,B 0.000,C 90.000,E1 147.661} C_DIS
LIN {X 0.149,Y -544.406,Z 1437.617,A 0.000,B 0.000,C 90.000,E1 147.041} C_DIS
LIN {X -0.020,Y -547.389,Z 1437.611,A 0.000,B 0.000,C 90.000,E1 145.928} C_DIS
LIN {X -0.196,Y -549.362,Z 1437.606,A 0.000,B 0.000,C 90.000,E1 145.102} C_DIS
LIN {X -0.091,Y -550.544,Z 1437.603,A 0.000,B 0.000,C 90.000,E1 144.529} C_DIS
LIN {X -0.239,Y -552.050,Z 1437.598,A 0.000,B 0.000,C 90.000,E1 143.703} C_DIS
LIN {X -0.048,Y -553.369,Z 1437.594,A 0.000,B 0.000,C 90.000,E1 142.844} C_DIS
LIN {X 0.156,Y -554.492,Z 1437.589,A 0.000,B 0.000,C 90.000,E1 141.984} C_DIS
LIN {X 0.009,Y -555.775,Z 1437.583,A 0.000,B 0.000,C 90.000,E1 140.884} C_DIS
LIN {X 0.311,Y -557.057,Z 1437.575,A 0.000,B 0.000,C 90.000,E1 139.461} C_DIS
LIN {X 0.215,Y -558.127,Z 1437.567,A 0.000,B 0.000,C 90.000,E1 138.081} C_DIS
LIN {X -0.201,Y -559.344,Z 1437.558,A 0.000,B 0.000,C 90.000,E1 136.458} C_DIS
LIN {X 0.049,Y -559.947,Z 1437.552,A 0.000,B 0.000,C 90.000,E1 135.324} C_DIS
LIN {X -0.021,Y -560.507,Z 1437.544,A 0.000,B 0.000,C 90.000,E1 133.947} C_DIS
LIN {X 0.321,Y -560.927,Z 1437.536,A 0.000,B 0.000,C 90.000,E1 132.528} C_DIS
LIN {X -0.170,Y -561.052,Z 1437.530,A 0.000,B 0.000,C 90.000,E1 131.472} C_DIS
LIN {X -0.198,Y -561.122,Z 1437.523,A 0.000,B 0.000,C 90.000,E1 130.092} C_DIS
LIN {X 0.196,Y -561.198,Z 1437.515,A 0.000,B 0.000,C 90.000,E1 128.669} C_DIS
LIN {X -0.105,Y -561.166,Z 1437.507,A 0.000,B 0.000,C 90.000,E1 127.317} C_DIS
LIN {X -0.069,Y -561.081,Z 1437.500,A 0.000,B 0.000,C 90.000,E1 125.931} C_DIS
LIN {X -0.140,Y -560.878,Z 1437.490,A 0.000,B 0.000,C 90.000,E1 124.278} C_DIS
LIN {X -0.206,Y -560.542,Z 1437.481,A 0.000,B 0.000,C 90.000,E1 122.625} C_DIS
LIN {X -0.140,Y -560.593,Z 1437.460,A 0.000,B 0.000,C 90.000,E1 118.743} C_DIS
LIN {X -0.037,Y -561.147,Z 1437.449,A 0.000,B 0.000,C 90.000,E1 116.796} C_DIS
LIN {X -0.023,Y -561.695,Z 1437.441,A 0.000,B 0.000,C 90.000,E1 115.412} C_DIS
LIN {X 0.013,Y -562.120,Z 1437.434,A 0.000,B 0.000,C 90.000,E1 114.027} C_DIS
LIN {X -0.217,Y -563.517,Z 1437.415,A 0.000,B 0.000,C 90.000,E1 110.737} C_DIS
LIN {X -0.272,Y -564.442,Z 1437.411,A 0.000,B 0.000,C 90.000,E1 110.066} C_DIS
LIN {X -0.314,Y -564.453,Z 1437.411,A 0.000,B 0.000,C 90.000,E1 110.066} C_DIS
LIN {X 0.029,Y -565.331,Z 1437.411,A 0.000,B 0.000,C 90.000,E1 109.885} C_DIS
LIN {X 0.060,Y -566.977,Z 1437.408,A 0.000,B 0.000,C 90.000,E1 109.504} C_DIS
LIN {X -0.011,Y -570.169,Z 1437.407,A 0.000,B 0.000,C 90.000,E1 109.214} C_DIS
LIN {X -0.225,Y -580.291,Z 1437.403,A 0.000,B 0.000,C 90.000,E1 108.598} C_DIS
LIN {X -0.320,Y -585.718,Z 1437.401,A 0.000,B 0.000,C 90.000,E1 108.181} C_DIS
LIN {X -0.058,Y -591.062,Z 1437.398,A 0.000,B 0.000,C 90.000,E1 107.692} C_DIS
LIN {X 0.184,Y -596.652,Z 1437.395,A 0.000,B 0.000,C 90.000,E1 107.040} C_DIS
LIN {X -0.177,Y -599.800,Z 1437.393,A 0.000,B 0.000,C 90.000,E1 106.677} C_DIS
LIN {X 0.111,Y -601.631,Z 1437.391,A 0.000,B 0.000,C 90.000,E1 106.386} C_DIS
LIN {X -0.225,Y -604.064,Z 1437.389,A 0.000,B 0.000,C 90.000,E1 106.024} C_DIS
LIN {X 0.084,Y -605.421,Z 1437.387,A 0.000,B 0.000,C 90.000,E1 105.733} C_DIS
LIN {X -0.237,Y -606.976,Z 1437.385,A 0.000,B 0.000,C 90.000,E1 105.371} C_DIS
LIN {X 0.244,Y -607.771,Z 1437.384,A 0.000,B 0.000,C 90.000,E1 105.064} C_DIS
LIN {X 0.310,Y -609.098,Z 1437.381,A 0.000,B 0.000,C 90.000,E1 104.537} C_DIS
LIN {X -0.203,Y -610.070,Z 1437.378,A 0.000,B 0.000,C 90.000,E1 104.064} C_DIS
LIN {X 0.229,Y -611.148,Z 1437.374,A 0.000,B 0.000,C 90.000,E1 103.244} C_DIS
LIN {X -0.269,Y -611.690,Z 1437.371,A 0.000,B 0.000,C 90.000,E1 102.771} C_DIS
LIN {X 0.184,Y -612.000,Z 1437.367,A 0.000,B 0.000,C 90.000,E1 101.951} C_DIS
LIN {X 0.288,Y -611.959,Z 1437.364,A 0.000,B 0.000,C 90.000,E1 101.422} C_DIS
LIN {X -0.212,Y -611.477,Z 1437.361,A 0.000,B 0.000,C 90.000,E1 100.950} C_DIS
LIN {X -0.116,Y -610.637,Z 1437.358,A 0.000,B 0.000,C 90.000,E1 100.423} C_DIS
LIN {X -0.134,Y -609.451,Z 1437.355,A 0.000,B 0.000,C 90.000,E1 99.905} C_DIS
LIN {X 0.208,Y -608.774,Z 1437.354,A 0.000,B 0.000,C 90.000,E1 99.613} C_DIS
LIN {X 0.184,Y -607.157,Z 1437.351,A 0.000,B 0.000,C 90.000,E1 99.095} C_DIS
LIN {X 0.244,Y -605.247,Z 1437.348,A 0.000,B 0.000,C 90.000,E1 98.568} C_DIS
LIN {X 0.018,Y -602.279,Z 1437.344,A 0.000,B 0.000,C 90.000,E1 97.936} C_DIS
LIN {X -0.239,Y -595.637,Z 1437.338,A 0.000,B 0.000,C 90.000,E1 96.777} C_DIS
LIN {X -0.154,Y -593.169,Z 1437.335,A 0.000,B 0.000,C 90.000,E1 96.372} C_DIS
LIN {X -0.278,Y -589.088,Z 1437.332,A 0.000,B 0.000,C 90.000,E1 95.853} C_DIS
LIN {X 0.113,Y -588.058,Z 1437.332,A 0.000,B 0.000,C 90.000,E1 95.682} C_DIS
LIN {X -0.227,Y -585.495,Z 1437.330,A 0.000,B 0.000,C 90.000,E1 95.448} C_DIS
LIN {X -0.038,Y -581.279,Z 1437.328,A 0.000,B 0.000,C 90.000,E1 95.049} C_DIS
LIN {X -0.026,Y -577.051,Z 1437.326,A 0.000,B 0.000,C 90.000,E1 94.702} C_DIS
LIN {X 0.097,Y -573.598,Z 1437.324,A 0.000,B 0.000,C 90.000,E1 94.359} C_DIS
LIN {X 0.057,Y -572.805,Z 1437.324,A 0.000,B 0.000,C 90.000,E1 94.245} C_DIS
LIN {X 0.234,Y -571.792,Z 1437.322,A 0.000,B 0.000,C 90.000,E1 93.955} C_DIS
LIN {X 0.021,Y -571.197,Z 1437.321,A 0.000,B 0.000,C 90.000,E1 93.841} C_DIS
LIN {X -0.061,Y -570.794,Z 1437.319,A 0.000,B 0.000,C 90.000,E1 93.440} C_DIS
LIN {X 0.070,Y -570.702,Z 1437.318,A 0.000,B 0.000,C 90.000,E1 93.154} C_DIS
LIN {X 0.018,Y -573.115,Z 1437.299,A 0.000,B 0.000,C 90.000,E1 89.885} C_DIS
LIN {X -0.274,Y -574.608,Z 1437.290,A 0.000,B 0.000,C 90.000,E1 88.282} C_DIS
LIN {X -0.099,Y -575.852,Z 1437.283,A 0.000,B 0.000,C 90.000,E1 86.906} C_DIS
LIN {X 0.134,Y -577.107,Z 1437.275,A 0.000,B 0.000,C 90.000,E1 85.527} C_DIS
LIN {X -0.181,Y -578.444,Z 1437.268,A 0.000,B 0.000,C 90.000,E1 84.204} C_DIS
LIN {X 0.169,Y -580.585,Z 1437.256,A 0.000,B 0.000,C 90.000,E1 82.008} C_DIS
LIN {X -0.253,Y -581.713,Z 1437.250,A 0.000,B 0.000,C 90.000,E1 80.971} C_DIS
LIN {X -0.109,Y -583.294,Z 1437.241,A 0.000,B 0.000,C 90.000,E1 79.342} C_DIS
LIN {X -0.058,Y -584.743,Z 1437.233,A 0.000,B 0.000,C 90.000,E1 77.993} C_DIS
LIN {X -0.224,Y -585.698,Z 1437.227,A 0.000,B 0.000,C 90.000,E1 76.937} C_DIS
LIN {X 0.010,Y -586.731,Z 1437.220,A 0.000,B 0.000,C 90.000,E1 75.574} C_DIS
LIN {X 0.264,Y -587.618,Z 1437.213,A 0.000,B 0.000,C 90.000,E1 74.212} C_DIS
LIN {X -0.041,Y -588.407,Z 1437.205,A 0.000,B 0.000,C 90.000,E1 72.906} C_DIS
LIN {X -0.168,Y -589.152,Z 1437.198,A 0.000,B 0.000,C 90.000,E1 71.583} C_DIS
LIN {X 0.014,Y -590.106,Z 1437.187,A 0.000,B 0.000,C 90.000,E1 69.699} C_DIS
LIN {X -0.121,Y -591.187,Z 1437.177,A 0.000,B 0.000,C 90.000,E1 67.847} C_DIS
LIN {X 0.104,Y -592.075,Z 1437.168,A 0.000,B 0.000,C 90.000,E1 66.230} C_DIS
LIN {X 0.044,Y -593.729,Z 1437.155,A 0.000,B 0.000,C 90.000,E1 63.845} C_DIS
LIN {X -0.061,Y -594.612,Z 1437.149,A 0.000,B 0.000,C 90.000,E1 62.794} C_DIS
LIN {X 0.055,Y -596.936,Z 1437.133,A 0.000,B 0.000,C 90.000,E1 59.871} C_DIS
LIN {X -0.154,Y -598.589,Z 1437.122,A 0.000,B 0.000,C 90.000,E1 58.043} C_DIS
LIN {X 0.037,Y -599.780,Z 1437.115,A 0.000,B 0.000,C 90.000,E1 56.707} C_DIS
LIN {X -0.274,Y -601.457,Z 1437.105,A 0.000,B 0.000,C 90.000,E1 54.895} C_DIS
LIN {X 0.034,Y -602.698,Z 1437.096,A 0.000,B 0.000,C 90.000,E1 53.290} C_DIS
LIN {X -0.018,Y -603.690,Z 1437.089,A 0.000,B 0.000,C 90.000,E1 51.984} C_DIS
LIN {X -0.267,Y -604.621,Z 1437.080,A 0.000,B 0.000,C 90.000,E1 50.436} C_DIS
LIN {X 0.041,Y -605.040,Z 1437.076,A 0.000,B 0.000,C 90.000,E1 49.622} C_DIS
LIN {X -0.052,Y -605.306,Z 1437.068,A 0.000,B 0.000,C 90.000,E1 48.324} C_DIS
LIN {X 0.076,Y -605.545,Z 1437.060,A 0.000,B 0.000,C 90.000,E1 46.743} C_DIS
LIN {X 0.212,Y -605.624,Z 1437.051,A 0.000,B 0.000,C 90.000,E1 45.162} C_DIS
LIN {X 0.296,Y -605.293,Z 1437.045,A 0.000,B 0.000,C 90.000,E1 44.109} C_DIS
LIN {X -0.239,Y -604.667,Z 1437.038,A 0.000,B 0.000,C 90.000,E1 42.852} C_DIS
LIN {X 0.064,Y -603.712,Z 1437.031,A 0.000,B 0.000,C 90.000,E1 41.515} C_DIS
LIN {X 0.151,Y -602.716,Z 1437.025,A 0.000,B 0.000,C 90.000,E1 40.458} C_DIS
LIN {X -0.376,Y -601.231,Z 1437.018,A 0.000,B 0.000,C 90.000,E1 39.197} C_DIS
LIN {X -0.103,Y -600.247,Z 1437.013,A 0.000,B 0.000,C 90.000,E1 38.382} C_DIS
LIN {X -0.205,Y -598.282,Z 1437.006,A 0.000,B 0.000,C 90.000,E1 37.076} C_DIS
LIN {X 0.134,Y -595.806,Z 1436.999,A 0.000,B 0.000,C 90.000,E1 35.724} C_DIS
LIN {X 0.084,Y -592.856,Z 1436.991,A 0.000,B 0.000,C 90.000,E1 34.405} C_DIS
LIN {X 0.181,Y -591.591,Z 1436.988,A 0.000,B 0.000,C 90.000,E1 33.865} C_DIS
LIN {X -0.138,Y -588.683,Z 1436.982,A 0.000,B 0.000,C 90.000,E1 32.832} C_DIS
LIN {X 0.123,Y -586.393,Z 1436.978,A 0.000,B 0.000,C 90.000,E1 32.005} C_DIS
LIN {X 0.178,Y -584.662,Z 1436.975,A 0.000,B 0.000,C 90.000,E1 31.465} C_DIS
LIN {X 0.085,Y -581.667,Z 1436.970,A 0.000,B 0.000,C 90.000,E1 30.669} C_DIS
LIN {X -0.034,Y -578.258,Z 1436.966,A 0.000,B 0.000,C 90.000,E1 29.873} C_DIS
LIN {X -0.116,Y -575.159,Z 1436.962,A 0.000,B 0.000,C 90.000,E1 29.205} C_DIS
LIN {X 0.189,Y -571.056,Z 1436.958,A 0.000,B 0.000,C 90.000,E1 28.359} C_DIS
LIN {X -0.231,Y -567.299,Z 1436.954,A 0.000,B 0.000,C 90.000,E1 27.719} C_DIS
LIN {X -0.012,Y -562.476,Z 1436.949,A 0.000,B 0.000,C 90.000,E1 26.873} C_DIS
LIN {X -0.063,Y -555.507,Z 1436.943,A 0.000,B 0.000,C 90.000,E1 25.771} C_DIS
LIN {X -0.112,Y -550.905,Z 1436.939,A 0.000,B 0.000,C 90.000,E1 25.079} C_DIS
LIN {X -0.077,Y -546.849,Z 1436.936,A 0.000,B 0.000,C 90.000,E1 24.515} C_DIS
LIN {X -0.072,Y -542.476,Z 1436.933,A 0.000,B 0.000,C 90.000,E1 23.951} C_DIS
LIN {X -0.097,Y -537.859,Z 1436.930,A 0.000,B 0.000,C 90.000,E1 23.387} C_DIS
LIN {X 0.194,Y -531.773,Z 1436.926,A 0.000,B 0.000,C 90.000,E1 22.642} C_DIS
LIN {X 0.110,Y -524.107,Z 1436.921,A 0.000,B 0.000,C 90.000,E1 21.791} C_DIS
LIN {X 0.182,Y -514.961,Z 1436.916,A 0.000,B 0.000,C 90.000,E1 20.791} C_DIS
LIN {X 0.065,Y -504.236,Z 1436.909,A 0.000,B 0.000,C 90.000,E1 19.685} C_DIS
LIN {X -0.131,Y -498.734,Z 1436.906,A 0.000,B 0.000,C 90.000,E1 19.141} C_DIS
LIN {X 0.188,Y -487.968,Z 1436.900,A 0.000,B 0.000,C 90.000,E1 18.000} C_DIS
LIN {X -0.037,Y -469.282,Z 1436.889,A 0.000,B 0.000,C 90.000,E1 16.024} C_DIS
LIN {X 0.152,Y -451.828,Z 1436.878,A 0.000,B 0.000,C 90.000,E1 14.008} C_DIS
LIN {X -0.044,Y -446.102,Z 1436.875,A 0.000,B 0.000,C 90.000,E1 13.411} C_DIS
LIN {X -0.075,Y -440.050,Z 1436.871,A 0.000,B 0.000,C 90.000,E1 12.827} C_DIS
LIN {X -0.026,Y -435.186,Z 1436.869,A 0.000,B 0.000,C 90.000,E1 12.411} C_DIS
LIN {X -0.124,Y -431.614,Z 1436.868,A 0.000,B 0.000,C 90.000,E1 12.175} C_DIS
LIN {X -0.022,Y -428.780,Z 1436.867,A 0.000,B 0.000,C 90.000,E1 12.007} C_DIS
LIN {X -0.111,Y -427.012,Z 1436.866,A 0.000,B 0.000,C 90.000,E1 11.951} C_DIS
LIN {X 0.060,Y -425.339,Z 1436.866,A 0.000,B 0.000,C 90.000,E1 11.895} C_DIS
LIN {X 0.099,Y -367.697,Z 1436.866,A 0.000,B 0.000,C 90.000,E1 11.883} C_DIS
LIN {X -0.145,Y -366.523,Z 1436.856,A 0.000,B 0.000,C 90.000,E1 10.018} C_DIS
LIN {X 0.061,Y -364.329,Z 1436.843,A 0.000,B 0.000,C 90.000,E1 7.757} C_DIS
LIN {X 0.035,Y -360.905,Z 1436.802,A 0.000,B 0.000,C 90.000,E1 0.286} C_DIS
LIN {X -0.053,Y -359.426,Z 1436.770,A 0.000,B 0.000,C 90.000,E1 354.546} C_DIS
LIN {X 0.070,Y -358.890,Z 1436.759,A 0.000,B 0.000,C 90.000,E1 352.648} C_DIS
LIN {X -0.020,Y -359.563,Z 1436.726,A 0.000,B 0.000,C 90.000,E1 346.645} C_DIS
LIN {X 0.001,Y -361.801,Z 1436.684,A 0.000,B 0.000,C 90.000,E1 339.135} C_DIS
LIN {X -0.154,Y -362.053,Z 1436.680,A 0.000,B 0.000,C 90.000,E1 338.411} C_DIS
LIN {X 0.189,Y -365.980,Z 1436.643,A 0.000,B 0.000,C 90.000,E1 331.641} C_DIS
LIN {X 0.029,Y -366.387,Z 1436.639,A 0.000,B 0.000,C 90.000,E1 330.923} C_DIS
LIN {X -0.031,Y -371.355,Z 1436.604,A 0.000,B 0.000,C 90.000,E1 324.642} C_DIS
LIN {X -0.043,Y -371.766,Z 1436.602,A 0.000,B 0.000,C 90.000,E1 324.276} C_DIS
LIN {X 0.013,Y -377.358,Z 1436.567,A 0.000,B 0.000,C 90.000,E1 318.038} C_DIS
LIN {X 0.012,Y -378.235,Z 1436.563,A 0.000,B 0.000,C 90.000,E1 317.310} C_DIS
LIN {X 0.002,Y -383.940,Z 1436.531,A 0.000,B 0.000,C 90.000,E1 311.515} C_DIS
LIN {X 0.088,Y -384.893,Z 1436.527,A 0.000,B 0.000,C 90.000,E1 310.782} C_DIS
LIN {X 0.262,Y -390.610,Z 1436.495,A 0.000,B 0.000,C 90.000,E1 305.025} C_DIS
LIN {X 0.106,Y -391.104,Z 1436.493,A 0.000,B 0.000,C 90.000,E1 304.692} C_DIS
LIN {X 0.022,Y -391.648,Z 1436.489,A 0.000,B 0.000,C 90.000,E1 303.992} C_DIS
LIN {X -0.080,Y -396.825,Z 1436.459,A 0.000,B 0.000,C 90.000,E1 298.693} C_DIS
LIN {X -0.210,Y -397.120,Z 1436.457,A 0.000,B 0.000,C 90.000,E1 298.359} C_DIS
LIN {X -0.055,Y -401.597,Z 1436.426,A 0.000,B 0.000,C 90.000,E1 292.717} C_DIS
LIN {X 0.222,Y -404.659,Z 1436.395,A 0.000,B 0.000,C 90.000,E1 287.094} C_DIS
LIN {X -0.079,Y -404.735,Z 1436.391,A 0.000,B 0.000,C 90.000,E1 286.441} C_DIS
LIN {X 0.214,Y -406.099,Z 1436.364,A 0.000,B 0.000,C 90.000,E1 281.535} C_DIS
LIN {X -0.176,Y -406.094,Z 1436.362,A 0.000,B 0.000,C 90.000,E1 281.243} C_DIS
LIN {X -0.097,Y -405.680,Z 1436.333,A 0.000,B 0.000,C 90.000,E1 276.024} C_DIS
LIN {X -0.165,Y -405.058,Z 1436.328,A 0.000,B 0.000,C 90.000,E1 274.992} C_DIS
LIN {X -0.060,Y -403.497,Z 1436.304,A 0.000,B 0.000,C 90.000,E1 270.802} C_DIS
LIN {X -0.092,Y -403.288,Z 1436.302,A 0.000,B 0.000,C 90.000,E1 270.458} C_DIS
LIN {X 0.091,Y -398.931,Z 1436.271,A 0.000,B 0.000,C 90.000,E1 264.837} C_DIS
LIN {X -0.040,Y -393.108,Z 1436.242,A 0.000,B 0.000,C 90.000,E1 259.567} C_DIS
LIN {X -0.079,Y -392.835,Z 1436.240,A 0.000,B 0.000,C 90.000,E1 259.218} C_DIS
LIN {X 0.034,Y -385.993,Z 1436.212,A 0.000,B 0.000,C 90.000,E1 254.212} C_DIS
LIN {X -0.026,Y -385.267,Z 1436.208,A 0.000,B 0.000,C 90.000,E1 253.504} C_DIS
LIN {X -0.004,Y -384.768,Z 1436.206,A 0.000,B 0.000,C 90.000,E1 253.142} C_DIS
LIN {X 0.221,Y -377.973,Z 1436.182,A 0.000,B 0.000,C 90.000,E1 248.773} C_DIS
LIN {X -0.044,Y -376.233,Z 1436.174,A 0.000,B 0.000,C 90.000,E1 247.358} C_DIS
LIN {X 0.057,Y -374.944,Z 1436.170,A 0.000,B 0.000,C 90.000,E1 246.613} C_DIS
LIN {X -0.208,Y -368.417,Z 1436.148,A 0.000,B 0.000,C 90.000,E1 242.615} C_DIS
LIN {X 0.097,Y -366.047,Z 1436.137,A 0.000,B 0.000,C 90.000,E1 240.717} C_DIS
LIN {X 0.004,Y -359.196,Z 1436.115,A 0.000,B 0.000,C 90.000,E1 236.628} C_DIS
LIN {X 0.021,Y -355.842,Z 1436.100,A 0.000,B 0.000,C 90.000,E1 233.989} C_DIS
LIN {X -0.173,Y -348.793,Z 1436.075,A 0.000,B 0.000,C 90.000,E1 229.461} C_DIS
LIN {X -0.097,Y -346.185,Z 1436.062,A 0.000,B 0.000,C 90.000,E1 227.148} C_DIS
LIN {X -0.088,Y -345.065,Z 1436.058,A 0.000,B 0.000,C 90.000,E1 226.377} C_DIS
LIN {X 0.094,Y -338.586,Z 1436.030,A 0.000,B 0.000,C 90.000,E1 221.310} C_DIS
LIN {X 0.094,Y -336.840,Z 1436.019,A 0.000,B 0.000,C 90.000,E1 219.358} C_DIS
LIN {X 0.014,Y -330.861,Z 1435.988,A 0.000,B 0.000,C 90.000,E1 213.865} C_DIS
LIN {X 0.149,Y -329.296,Z 1435.975,A 0.000,B 0.000,C 90.000,E1 211.465} C_DIS
LIN {X -0.154,Y -324.669,Z 1435.942,A 0.000,B 0.000,C 90.000,E1 205.540} C_DIS
LIN {X 0.174,Y -323.837,Z 1435.928,A 0.000,B 0.000,C 90.000,E1 203.078} C_DIS
LIN {X -0.017,Y -321.124,Z 1435.881,A 0.000,B 0.000,C 90.000,E1 194.662} C_DIS
LIN {X 0.138,Y -320.932,Z 1435.877,A 0.000,B 0.000,C 90.000,E1 193.828} C_DIS
LIN {X -0.076,Y -321.562,Z 1435.832,A 0.000,B 0.000,C 90.000,E1 185.796} C_DIS
LIN {X -0.143,Y -324.415,Z 1435.790,A 0.000,B 0.000,C 90.000,E1 178.165} C_DIS
LIN {X -0.141,Y -325.376,Z 1435.783,A 0.000,B 0.000,C 90.000,E1 176.963} C_DIS
LIN {X -0.100,Y -329.112,Z 1435.750,A 0.000,B 0.000,C 90.000,E1 170.971} C_DIS
LIN {X -0.171,Y -334.238,Z 1435.726,A 0.000,B 0.000,C 90.000,E1 166.645} C_DIS
LIN {X 0.134,Y -361.903,Z 1435.726,A 0.000,B 0.000,C 90.000,E1 166.589} C_DIS
LIN {X 0.041,Y -364.674,Z 1435.725,A 0.000,B 0.000,C 90.000,E1 166.533} C_DIS
END
